IF etDiag <> GD.ET_Diag.Ok AND NOT xUpdateStructsException THEN
	xUpdateStructsException := TRUE;
	
	stUpdateStructsException.sMsg := PDL.FC_MultiConcat(i_sString1 := 'Update AddInterface: Nocke1 - ', 
														i_sString2 := GD.FC_EtDiagToString(i_etDiag := etDiag), 
														i_sString3 := ' - ', 
														i_sString4 := FC_EtDiagExtExampleLeafModuleToString(i_etDiagExt := etDiagExtExampleLeaf));
END_IF	

(*****************************************************************************************************************************************************)
(* Update ILS Data *)

// stSlave3Interface.stEndless.pstIlsData	:= ADR(G_stIlsData);
// stSlave3Interface.stMultiCam.pstIlsData	:= ADR(G_stIlsData);

// stSlave4Interface.stEndless.pstIlsData	:= ADR(G_stIlsData);
// stSlave4Interface.stMultiCam.pstIlsData	:= ADR(G_stIlsData);

(*****************************************************************************************************************************************************)
(* Set exception if any exception occurred *)

fbExceptionHandler.SetException(i_xExceptionActive	:= xUpdateStructsException, 
								iq_stException		:= stUpdateStructsException, 
								iq_stExceptionList	:= iq_stExceptionList);
					
xInitSuccessful := xInitSuccessful AND NOT xUpdateStructsException;

etDiag := GD.ET_Diag.Ok;	
(* End of system generated code, could be modified for your application *)
END_ACTION

END_PROGRAM

// LMC_PacDrive/Application/FB_ExampleLeafModule
FUNCTION_BLOCK FB_ExampleLeafModule

VAR_IN_OUT
(* TPL.ST_StandardModuleInterface *)	
	iq_stStandardModuleItf			: TPL.ST_StandardModuleInterface;
	
(* ExceptionHandling and Logging *)	
	iq_stExceptionList				: TPL.ST_ExceptionList;
	iq_stLogDataList				: TPL.ST_LogDataList;
	
(* ST_ExampleLeafModuleInterface *)
	iq_stExampleLeafModuleItf		: ST_ExampleLeafModuleInterface;
END_VAR

VAR
	xEnableFlag : BOOL;
	
	udii : UDINT;
	
	xInitHomingDone : BOOL;
	xNotAbleToSetException : BOOL;

	etDiagBuffer		: GD.ET_Diag;
	etDiagExtBufferTPL	: TPL.ET_DiagExt;
	sDiagMsgBuffer		: STRING[80];
	
	xDiagQuitFlag : BOOL;
	
	
	xExceptionReactionOutsideRange		: BOOL;
	
	stExceptionInit						: TPL.ST_Exception;
	stExceptionCmdImpossibleState		: TPL.ST_Exception;
	stExceptionCmdUnknown				: TPL.ST_Exception;
	stExceptionCmdImpossibleOverwrite	: TPL.ST_Exception;
	stWarningCmdImpossibleReaction		: TPL.ST_Exception;
	stExceptionHoming					: TPL.ST_Exception;
	stExceptionModuleReaction1			: TPL.ST_Exception;
	stExceptionModuleReaction2			: TPL.ST_Exception;
	stExceptionModuleReaction3			: TPL.ST_Exception;
	stExceptionModuleReaction4			: TPL.ST_Exception;
	stExceptionDriveFatal				: TPL.ST_Exception;
	stExcepitonDrive					: TPL.ST_Exception;
	stWarningDrive						: TPL.ST_Exception;

	stModuleReaction			: TPL.ST_Reaction;
	stLocalReaction				: TPL.ST_Reaction;
	stEmptyReaction				: TPL.ST_Reaction;
	stReaction1					: TPL.ST_Reaction;
	stReaction2					: TPL.ST_Reaction;
	stReaction3					: TPL.ST_Reaction;
	stReaction4					: TPL.ST_Reaction;

	udiDoSomethingCounter	: UDINT := 0;

	xCheckCmdException	: BOOL;
	xOpModeCmd			: BOOL;
	xCommandRefused		: BOOL;

	(* OpMode enable and active flags *)
	xHomingEnable : BOOL;
	xHomingActive : BOOL;
	xAutoEnable : BOOL;
	xAutoActive : BOOL;

	xCommandAcceptedInThisCycle : BOOL;

	xHomingException : BOOL;

	xRandomExceptionTrigger: BOOL;

	xStartFlag : BOOL;

	fbLogger : TPL.FB_Logger;
	fbLoggerPoint	: APL.FB_LoggerPoint;
	
	etStateOld : ET_ExampleLeafModuleState;
	udiMyResultSource : UDINT;
	
	ifRefActualValuesPosition : SystemConfigurationItf.IF_RefActualValuesPosition; 
	xSuccess : BOOL;
END_VAR

VAR CONSTANT
	c_udiDoSomeThingLevel : UDINT := 500;
END_VAR

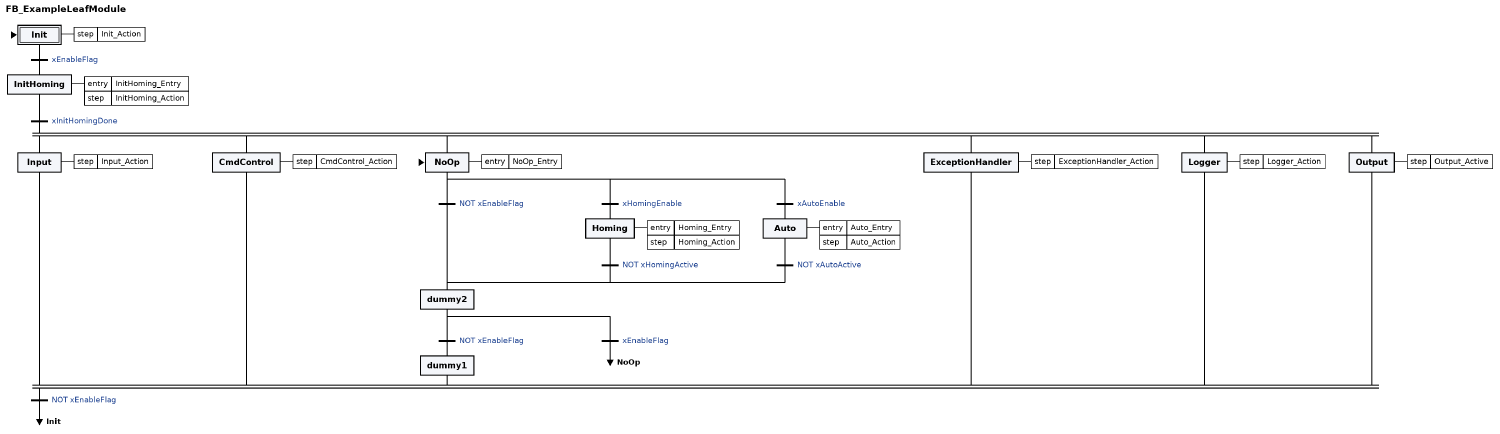
INITIAL_STEP Init:
    Init_Action(N);  // step action
END_STEP
TRANSITION FROM Init TO InitHoming
    := xEnableFlag;
END_TRANSITION
STEP InitHoming:
    InitHoming_Entry(P1);  // entry action
    InitHoming_Action(N);  // step action
END_STEP
TRANSITION FROM InitHoming TO (Input, CmdControl, NoOp, ExceptionHandler, Logger, Output)
    := xInitHomingDone;
END_TRANSITION
STEP Input:
    Input_Action(N);  // step action
END_STEP
STEP CmdControl:
    CmdControl_Action(N);  // step action
END_STEP
STEP NoOp:
    NoOp_Entry(P1);  // entry action
END_STEP
TRANSITION FROM NoOp TO dummy2
    := NOT xEnableFlag;
END_TRANSITION
TRANSITION FROM NoOp TO Homing
    := xHomingEnable;
END_TRANSITION
STEP Homing:
    Homing_Entry(P1);  // entry action
    Homing_Action(N);  // step action
END_STEP
TRANSITION FROM Homing TO dummy2
    := NOT xHomingActive;
END_TRANSITION
TRANSITION FROM NoOp TO Auto
    := xAutoEnable;
END_TRANSITION
STEP Auto:
    Auto_Entry(P1);  // entry action
    Auto_Action(N);  // step action
END_STEP
TRANSITION FROM Auto TO dummy2
    := NOT xAutoActive;
END_TRANSITION
STEP dummy2:
END_STEP
TRANSITION FROM dummy2 TO dummy1
    := NOT xEnableFlag;
END_TRANSITION
TRANSITION FROM dummy2 TO NoOp
    := xEnableFlag;
END_TRANSITION
STEP dummy1:
END_STEP
STEP ExceptionHandler:
    ExceptionHandler_Action(N);  // step action
END_STEP
STEP Logger:
    Logger_Action(N);  // step action
END_STEP
STEP Output:
    Output_Active(N);  // step action
END_STEP
TRANSITION FROM (Input, CmdControl, dummy1, ExceptionHandler, Logger, Output) TO Init
    := NOT xEnableFlag;
END_TRANSITION

ACTION Auto_Action:
(* Start application code *)
IF(iq_stExampleLeafModuleItf.q_etState = ET_ExampleLeafModuleState.AutoWaitForStart) THEN
	IF(xAutoEnable) THEN
		IF(xStartFlag) THEN
			iq_stExampleLeafModuleItf.q_etState := ET_ExampleLeafModuleState.AutoRunning;
		END_IF
	ELSE
		xAutoActive := FALSE;
	END_IF
END_IF

IF(NOT xStartFlag AND iq_stExampleLeafModuleItf.q_etState = ET_ExampleLeafModuleState.AutoRunning) THEN
	iq_stExampleLeafModuleItf.q_etState := ET_ExampleLeafModuleState.AutoWaitForStart;
END_IF

IF(iq_stExampleLeafModuleItf.q_etState = ET_ExampleLeafModuleState.AutoRunning) THEN
	IF(xAutoEnable) THEN
		iq_stExampleLeafModuleItf.q_xValue := ifRefActualValuesPosition.RefPosition >= iq_stExampleLeafModuleItf.i_lrPosMin AND 
													ifRefActualValuesPosition.RefPosition <= iq_stExampleLeafModuleItf.i_lrPosMax;
	ELSE
		iq_stExampleLeafModuleItf.q_etState := ET_ExampleLeafModuleState.AutoWaitForStart;
	END_IF
END_IF
(* End application code *)
END_ACTION

ACTION Auto_Entry:
iq_stExampleLeafModuleItf.q_etState := ET_ExampleLeafModuleState.AutoWaitForStart;
xAutoActive := TRUE;
END_ACTION

METHOD CancelException
VAR_IN_OUT
	iq_stException	: TPL.ST_Exception;
END_VAR
TPL.FC_SetException(	i_xExceptionActive	:= FALSE,
						iq_stException		:= iq_stException,
						iq_stExceptionList	:= iq_stExceptionList,
						iq_stLogDataList	:= iq_stLogDataList,
						q_etDiag 			=> etDiagBuffer,
						q_etDiagExt 		=> etDiagExtBufferTPL,
						q_sMsg 				=> sDiagMsgBuffer);
END_METHOD

ACTION CheckCmd:
(*--------------------------------------------------------------------------------------------------*)
(* CheckCMD is checking if CMD is supported by this module *)
(*--------------------------------------------------------------------------------------------------*)
xOpModeCMD			:= FALSE;
xCheckCmdException	:= FALSE;

IF 	iq_stStandardModuleItf.iq_diCMD = ET_ExampleLeafModuleCmd.Homing OR
	iq_stStandardModuleItf.iq_diCMD = ET_ExampleLeafModuleCmd.Auto OR
	iq_stStandardModuleItf.iq_diCMD = ET_ExampleLeafModuleCmd.Stop THEN

	xOpModeCMD := TRUE;
ELSIF iq_stStandardModuleItf.iq_diCMD = ET_ExampleLeafModuleCmd.Start OR
	  iq_stStandardModuleItf.iq_diCMD = ET_ExampleLeafModuleCmd.Hold THEN
	;
ELSE
	xCheckCmdException := TRUE;
END_IF
END_ACTION

ACTION CmdControl_Action:
(* CMD execution

	algorithm:
	----------

	detect new command?
		check command?
			execute command;
		end
	end

	is command running (at least one cycle)?	
		is command finished?
			signal success/unsuccessful
		end
	end
*)

xCommandAcceptedInThisCycle := FALSE;

(* Detect new command *)
IF(iq_stStandardModuleItf.i_xEnable) THEN
	IF (iq_stStandardModuleItf.iq_diCMD > 0 AND (NOT iq_stStandardModuleItf.q_xCMDActive (* In case no command is active *)
			OR iq_stStandardModuleItf.iq_diCMD <> iq_stStandardModuleItf.q_diCMDActive) (* In case a command is active *)) THEN
	
		xCommandRefused := FALSE; (* Flag is set by RefuseCommand() action *)
	
		(* Check command *)
		CheckCmd();
		IF(xCheckCmdException) THEN
			(*** Check for unknown command ***)
			stExceptionCmdUnknown.sMsg := Standard.CONCAT('Cmd unknown: ',DINT_TO_STRING(iq_stStandardModuleItf.iq_diCmd));
			ReportException(iq_stException := stExceptionCmdUnknown); 
			RefuseCommand();
		ELSE
			(*** Check for impossible overwrite ***)
			IF(iq_stStandardModuleItf.q_xCMDActive AND iq_stStandardModuleItf.iq_diCMD <> ET_ExampleLeafModuleCmd.Stop) THEN (* In this module only the ET_ExampleLeafModuleCmd.Stop command can overwrite other commands *)
				stExceptionCmdImpossibleOverwrite.sMsg := PDL.FC_MultiConcat(	i_sString1 := 'Cmd impossible: ',
																				i_sString2 := FC_EtExampleLeafModuleCmdToString(i_diCmd := iq_stStandardModuleItf.iq_diCmd),
																				i_sString3 := '; Cmd active: ',
																				i_sString4 := FC_EtExampleLeafModuleCmdToString(i_diCmd := iq_stStandardModuleItf.q_diCmdActive) );
				ReportException(iq_stException := stExceptionCmdImpossibleOverwrite);	
				RefuseCommand();
			ELSE
				(*** Check for impossible state ***)
				IF(NOT xOpModeCmd AND (* In this module, all OpMode commands are always possible independent of the state *)
					(iq_stExampleLeafModuleItf.q_etState = ET_ExampleLeafModuleState.NoOp (* Start and Hold are not possible in NoOp *)
					OR (iq_stExampleLeafModuleItf.q_etState = ET_ExampleLeafModuleState.HomingWaitForStart OR iq_stExampleLeafModuleItf.q_etState = ET_ExampleLeafModuleState.HomingDone) AND iq_stStandardModuleItf.iq_diCMD = ET_ExampleLeafModuleCmd.Hold) (* Hold is not supported in homing *)
					) THEN
					stExceptionCmdImpossibleState.sMsg := PDL.FC_MultiConcat(	i_sString1 := 'Cmd impossible: ',
																				i_sString2 := FC_EtExampleLeafModuleCmdToString(i_diCmd := iq_stStandardModuleItf.iq_diCmd),
																				i_sString3 := '; State: ',
																				i_sString4 := FC_EtExampleLeafModuleStateToString(i_etState := iq_stExampleLeafModuleItf.q_etState) );
					ReportException(iq_stException := stExceptionCmdImpossibleState);
					RefuseCommand();
				ELSE
					(* Check for impossible commands due to active error reactions *)
					IF	iq_stStandardModuleItf.iq_diCMD = ET_ExampleLeafModuleCmd.Start 
							AND (stModuleReaction.axReaction[TPL.ET_Reaction.AsyncStop] OR 
								 stModuleReaction.axReaction[TPL.ET_Reaction.SyncStopEH] OR 
								 stModuleReaction.axReaction[TPL.ET_Reaction.SyncStopEL] OR 
								 stModuleReaction.axReaction[TPL.ET_Reaction.StopEndOfCycle]) (* Start impossible if error reaction 4 or higher *)
						OR 
						
						iq_stStandardModuleItf.iq_diCMD <> ET_ExampleLeafModuleCmd.Stop 
							AND (stModuleReaction.axReaction[TPL.ET_Reaction.AsyncStop] OR 
								 stModuleReaction.axReaction[TPL.ET_Reaction.SyncStopEH] OR 
								 stModuleReaction.axReaction[TPL.ET_Reaction.SyncStopEL]) THEN (* Everything else, with exception of Stop, impossible if error reaction 3 or higher *)

						stWarningCmdImpossibleReaction.sMsg := PDL.FC_MultiConcat(	i_sString1 := 'Cmd impossible: ',
																					i_sString2 := FC_EtExampleLeafModuleCmdToString(i_diCmd := iq_stStandardModuleItf.iq_diCmd),
																					i_sString3 := '; Reaction: ',
																					i_sString4 := TPL.FC_GetStandardReactionName(iq_stReaction := stModuleReaction));
						ReportException(iq_stException := stWarningCmdImpossibleReaction);
						RefuseCommand();
					END_IF
				END_IF
			END_IF
		END_IF
	
		IF(NOT xCommandRefused) THEN (* Command has passed all checks, execute command *)
			IF fbLoggerPoint.etLogLevel >= APL.ET_LogLevel.UserAction THEN
				fbLoggerPoint.AddLogEntry(	i_etLogLevel	:= APL.ET_LogLevel.UserAction,
											i_etDiag		:= GD.ET_Diag.Ok,
											i_udiDiagExt	:= ET_DiagExtExampleLeafModule.Ok,
											i_sMessage		:= Standard.CONCAT(Standard.CONCAT(Standard.CONCAT('Command executing: ', FC_etExampleLeafModuleCmdToString(i_diCmd := iq_stStandardModuleItf.iq_diCmd)),' number: '),DINT_TO_STRING(iq_stStandardModuleItf.iq_diCmd)),
											q_etDiag		:= ,
											q_etDiagExt		:= );
			END_IF
			(* Accept command *)
			iq_stStandardModuleItf.q_xCMDActive := TRUE;
			iq_stStandardModuleItf.q_xCMDDone := FALSE;
			iq_stStandardModuleItf.q_diCMDActive := iq_stStandardModuleItf.iq_diCMD;
	
			xCommandAcceptedInThisCycle := TRUE; (* Signal for command done checks *)
	
			IF(xOpModeCMD) THEN
				DisableAllJobs();
				
				CASE iq_stStandardModuleItf.iq_diCMD OF
					ET_ExampleLeafModuleCmd.Stop:
						;	(* Do nothing, disabled OpMode flags automatically lead to NoOp *)
						
					ET_ExampleLeafModuleCmd.Homing:
						xHomingEnable := TRUE;
					
					ET_ExampleLeafModuleCmd.Auto:
						xAutoEnable := TRUE;
				END_CASE
			ELSE
				(* Action commands *)
				CASE iq_stStandardModuleItf.iq_diCMD OF
					ET_ExampleLeafModuleCmd.Start:
						xStartFlag := TRUE;
					
					ET_ExampleLeafModuleCmd.Hold:
						xStartFlag := FALSE;
				END_CASE
			END_IF
		END_IF (* New command? *)
	END_IF

(********************************************* Check successful and unsucessful of given commands ****************************************)

	(* Check if active command is done or is stopped by an error *)
	IF(NOT xCommandAcceptedInThisCycle) THEN (* Don't execute these checks if we accepted a new command in this cycle
		to ensure that execution of every command requires a minimum of 2 cycles *)

		IF(iq_stStandardModuleItf.q_xCMDActive) THEN
			CASE iq_stStandardModuleItf.iq_diCmd OF
				ET_ExampleLeafModuleCmd.Homing:
					(* Successful *)
					IF(xHomingActive) THEN
						SignalSuccessfulExecution();
					END_IF
					(* Unsucessful *)
					IF (stModuleReaction.axReaction[TPL.ET_Reaction.AsyncStop] OR 
						stModuleReaction.axReaction[TPL.ET_Reaction.SyncStopEL] OR 
						stModuleReaction.axReaction[TPL.ET_Reaction.SyncStopEH]) THEN
						
						SignalUnsuccessfulExecution();
					END_IF
					
				ET_ExampleLeafModuleCmd.Auto:
					(* Successful *)
					IF(xAutoActive) THEN
						SignalSuccessfulExecution();
					END_IF
					(* Unsucessful *)
					IF (stModuleReaction.axReaction[TPL.ET_Reaction.AsyncStop] OR 
						stModuleReaction.axReaction[TPL.ET_Reaction.SyncStopEL] OR 
						stModuleReaction.axReaction[TPL.ET_Reaction.SyncStopEH]) THEN

						SignalUnsuccessfulExecution();
					END_IF
	
				ET_ExampleLeafModuleCmd.Stop:
					(* Successful *)
					IF(iq_stExampleLeafModuleItf.q_etState = ET_ExampleLeafModuleState.NoOp) THEN
						SignalSuccessfulExecution();
					END_IF
					
				ET_ExampleLeafModuleCmd.Start:
					IF(iq_stExampleLeafModuleItf.q_etState = ET_ExampleLeafModuleState.HomingDone) THEN
						xStartFlag := FALSE;
					END_IF
					(* Successful *)
					IF(iq_stExampleLeafModuleItf.q_etState = ET_ExampleLeafModuleState.HomingDone AND NOT xHomingException
						OR iq_stExampleLeafModuleItf.q_etState = ET_ExampleLeafModuleState.AutoRunning) THEN
						SignalSuccessfulExecution();
					END_IF
					(* Unsucessful *)
					IF (stModuleReaction.axReaction[TPL.ET_Reaction.AsyncStop] OR 
						stModuleReaction.axReaction[TPL.ET_Reaction.SyncStopEL] OR 
						stModuleReaction.axReaction[TPL.ET_Reaction.SyncStopEH] OR 
						stModuleReaction.axReaction[TPL.ET_Reaction.StopEndOfCycle]  OR
						iq_stExampleLeafModuleItf.q_etState = ET_ExampleLeafModuleState.HomingDone AND xHomingException) THEN
						
						SignalUnsuccessfulExecution();
					END_IF
					
				ET_ExampleLeafModuleCmd.Hold:
					(* Successful *)
					IF(iq_stExampleLeafModuleItf.q_etState = ET_ExampleLeafModuleState.AutoWaitForStart) THEN
						SignalSuccessfulExecution();
					END_IF
					(* Unsucessful *)
					IF (stModuleReaction.axReaction[TPL.ET_Reaction.AsyncStop] OR 
						stModuleReaction.axReaction[TPL.ET_Reaction.SyncStopEL] OR 
						stModuleReaction.axReaction[TPL.ET_Reaction.SyncStopEH]) THEN

						SignalUnsuccessfulExecution();
					END_IF
			END_CASE
		END_IF
	END_IF
ELSE
	(* Module is going to be disabled *)
	iq_stStandardModuleItf.q_xReady := FALSE;
	xEnableFlag := FALSE;
	
	DisableAllJobs();
	
	xStartFlag := FALSE;

	IF(iq_stStandardModuleItf.q_xCmdActive) THEN (* If a command is currently active, cancel its execution *)
		SignalUnsuccessfulExecution();
	ELSE
		InactiveCmdExecution(); (* Command processing as if we were disabled *)
	END_IF
END_IF
END_ACTION

ACTION DiagQuit:
IF(iq_stStandardModuleItf.i_xDiagQuit AND NOT xDiagQuitFlag) THEN
	(* Rising edge of error quit *)
	xDiagQuitFlag := TRUE;
	xNotAbleToSetException := FALSE;

	FOR udii := 1 TO TPL.ET_Reaction.MainsContactorOff DO
		stLocalReaction.axReaction[udii] := FALSE;
	END_FOR

	iq_stStandardModuleItf.q_etDiag := GD.ET_Diag.Ok;

	IF(iq_stStandardModuleItf.iq_diCMD < 0) THEN
		iq_stStandardModuleItf.iq_diCMD := 0;
	END_IF
	IF fbLoggerPoint.etLogLevel >= APL.ET_LogLevel.UserAction THEN
		fbLoggerPoint.AddLogEntry(	i_etLogLevel	:= APL.ET_LogLevel.UserAction,
									i_etDiag		:= GD.ET_Diag.Ok,
									i_udiDiagExt	:= ET_DiagExtExampleLeafModule.Ok,
									i_sMessage		:= 'Diag Quit',
									q_etDiag		:= ,
									q_etDiagExt		:= );
	END_IF
ELSIF(NOT iq_stStandardModuleItf.i_xDiagQuit AND xDiagQuitFlag) THEN
	xDiagQuitFlag := FALSE;
END_IF
END_ACTION

ACTION DisableAllJobs:
(* Disable current OpMode and enable next one *)
xHomingEnable := FALSE;
xAutoEnable := FALSE;

xStartFlag := FALSE; (* On OpMode change, always reset the start flag *)
END_ACTION

ACTION Homing_Entry:
iq_stExampleLeafModuleItf.q_etState := ET_ExampleLeafModuleState.HomingWaitForStart;
xHomingActive := TRUE;


(* Start application code *)
udiDoSomethingCounter := 0;
(* End application code *)
END_ACTION

ACTION InactiveCmdExecution:
(* Command execution if module is not active (q_xActive = FALSE) or currently deactivating (i_xEnable = FALSE, q_xActive is still TRUE) *)
IF iq_stStandardModuleItf.iq_diCmd <> 0 THEN
	IF(NOT iq_stStandardModuleItf.i_xEnable) THEN
		iq_stStandardModuleItf.iq_diCmd := 0; (* All commands are signaled executed if module is disabled *)
(*ELSE*)
	ELSIF(iq_stStandardModuleItf.iq_diCmd > 0) THEN (* New command *)
		(* Command execution during enable but module is not ready for commands yet ==> error *)
		//xExceptionCmdImpossibleState := TRUE;

		stExceptionCmdImpossibleState.sMsg := PDL.FC_MultiConcat(	i_sString1 := 'Cmd impossible: ',
																	i_sString2 := FC_EtExampleLeafModuleCmdToString(i_diCmd := ABS(iq_stStandardModuleItf.iq_diCmd)),
																	i_sString3 := '; State: ',
																	i_sString4 := FC_EtExampleLeafModuleStateToString(i_etState := iq_stExampleLeafModuleItf.q_etState));
		ReportException(iq_stException := stExceptionCmdImpossibleState);
		iq_stStandardModuleItf.iq_diCmd:= - ABS(iq_stStandardModuleItf.iq_diCmd);
	END_IF
END_IF
iq_stStandardModuleItf.q_xCmdActive := FALSE;
iq_stStandardModuleItf.q_xCmdDone := FALSE;
iq_stStandardModuleItf.q_diCmdActive := 0;
END_ACTION

ACTION Init_Action:
iq_stStandardModuleItf.q_xActive			:= FALSE;
iq_stStandardModuleItf.q_xReady				:= FALSE;

iq_stStandardModuleItf.q_etDiag				:= GD.ET_Diag.Ok;
iq_stStandardModuleItf.q_udiDiagExt			:= ET_DiagExtExampleLeafModule.Disabled;
iq_stStandardModuleItf.q_sDiagExt			:= FC_EtDiagExtExampleLeafModuleToString(i_etDiagExt := iq_stStandardModuleItf.q_udiDiagExt);
iq_stStandardModuleItf.q_sMsg				:= '';

iq_stStandardModuleItf.q_dwModuleType		:= ET_ModuleType.ExampleLeafModule;
iq_stStandardModuleItf.q_sModuleTypeName	:= 'ExampleLeafModule';
iq_stStandardModuleItf.q_udiModuleVersion	:= 1;

iq_stExampleLeafModuleItf.q_etState	:= ET_ExampleLeafModuleState.Disabled;

THIS^.DiagQuit();
THIS^.InactiveCmdExecution();

udiMyResultSource := ET_ExceptionSource.ExampleLeafModule; (* Has to be coded this way to get around compiler restrictions*)

(* detect invalid configurations and avoid array index out of range error *)
IF(iq_stStandardModuleItf.iq_stExt.udiReactionOffset + TPL. ET_Reaction.MainsContactorOff > TPL.Gc_udiMaxNumberOfReactions) OR xExceptionReactionOutsideRange THEN (* module uses error reactions 1 to 5 *)
	xExceptionReactionOutsideRange := TRUE; (* create unquittable error *)
	
	(* create exception *)
	stExceptionInit.etDiag					:= GD.ET_Diag.InputParameterInvalid;
	stExceptionInit.udiDiagExt				:= ET_DiagExtExampleLeafModule.ReactionOffsetRange;
	stExceptionInit.sMsg					:= Standard.CONCAT('Value: ', UDINT_TO_STRING(iq_stStandardModuleItf.iq_stExt.udiReactionOffset));
	stExceptionInit.udiModuleId				:= iq_stStandardModuleItf.i_udiModuleId;
	stExceptionInit.sModuleName				:= iq_stStandardModuleItf.i_sModuleName;
	stExceptionInit.etSource				:= udiMyResultSource;
	stExceptionInit.timDelayTime			:= T#0MS;
	stExceptionInit.wHmiAttributes			:= 0;
	stExceptionInit.xAutoQuit				:= FALSE;
	stExceptionInit.stReaction.axReaction[TPL.ET_Reaction.AsyncStop]	:= TRUE; (* without offset on purpose *)
	
	iq_stStandardModuleItf.iq_stExt.udiReactionOffset := 0;
	
	ReportException(iq_stException := stExceptionInit);
ELSIF (iq_stStandardModuleItf.i_xEnable) THEN
	stReaction1 := stEmptyReaction;
	stReaction1.axReaction[iq_stStandardModuleItf.iq_stExt.udiReactionOffset + TPL.ET_Reaction.AsyncStop] := TRUE;
	stReaction2 := stEmptyReaction;
	stReaction2.axReaction[iq_stStandardModuleItf.iq_stExt.udiReactionOffset + TPL.ET_Reaction.SyncStopEL] := TRUE;
	stReaction3 := stEmptyReaction;
	stReaction3.axReaction[iq_stStandardModuleItf.iq_stExt.udiReactionOffset + TPL.ET_Reaction.SyncStopEH] := TRUE;
	stReaction4 := stEmptyReaction;
	stReaction4.axReaction[iq_stStandardModuleItf.iq_stExt.udiReactionOffset + TPL.ET_Reaction.StopEndOfCycle] := TRUE;
	
	(* Initialization of exception structures *)
	stExceptionCmdUnknown.etDiag						:= GD.ET_Diag.ExecutionAborted;
	stExceptionCmdUnknown.udiDiagExt					:= ET_DiagExtExampleLeafModule.CmdUnknown;
	stExceptionCmdUnknown.sMsg							:= 'Command unknown'; (* Replaced on usage *)
	stExceptionCmdUnknown.udiModuleId					:= iq_stStandardModuleItf.i_udiModuleId;
	stExceptionCmdUnknown.sModuleName					:= iq_stStandardModuleItf.i_sModuleName;
	stExceptionCmdUnknown.etSource						:= udiMyResultSource;
	stExceptionCmdUnknown.timDelayTime					:= T#0MS;
	stExceptionCmdUnknown.wHmiAttributes				:= 0;
	stExceptionCmdUnknown.xAutoQuit						:= FALSE;
	stExceptionCmdUnknown.stReaction					:= stReaction1;

	stExceptionCmdImpossibleOverwrite.etDiag			:= GD.ET_Diag.ExecutionAborted;
	stExceptionCmdImpossibleOverwrite.udiDiagExt		:= ET_DiagExtExampleLeafModule.CmdImpossibleOverwrite;
	stExceptionCmdImpossibleOverwrite.sMsg				:= 'Impossible command overwrite'; (* Replaced on usage *)
	stExceptionCmdImpossibleOverwrite.udiModuleId		:= iq_stStandardModuleItf.i_udiModuleId;
	stExceptionCmdImpossibleOverwrite.sModuleName		:= iq_stStandardModuleItf.i_sModuleName;
	stExceptionCmdImpossibleOverwrite.etSource			:= udiMyResultSource;
	stExceptionCmdImpossibleOverwrite.timDelayTime		:= T#0MS;
	stExceptionCmdImpossibleOverwrite.wHmiAttributes	:= 0;
	stExceptionCmdImpossibleOverwrite.xAutoQuit			:= FALSE;
	stExceptionCmdImpossibleOverwrite.stReaction		:= stReaction1;
	
	stExceptionCmdImpossibleState.etDiag				:= GD.ET_Diag.ExecutionAborted;
	stExceptionCmdImpossibleState.udiDiagExt			:= ET_DiagExtExampleLeafModule.CmdImpossibleState;
	stExceptionCmdImpossibleState.sMsg					:= 'Impossible command for state'; (* Replaced on usage *)
	stExceptionCmdImpossibleState.udiModuleId			:= iq_stStandardModuleItf.i_udiModuleId;
	stExceptionCmdImpossibleState.sModuleName			:= iq_stStandardModuleItf.i_sModuleName;
	stExceptionCmdImpossibleState.etSource				:= udiMyResultSource;
	stExceptionCmdImpossibleState.timDelayTime			:= T#0MS;
	stExceptionCmdImpossibleState.wHmiAttributes		:= 0;
	stExceptionCmdImpossibleState.xAutoQuit				:= FALSE;
	stExceptionCmdImpossibleState.stReaction			:= stReaction1;

	stWarningCmdImpossibleReaction.etDiag				:= GD.ET_Diag.ExecutionAborted;
	stWarningCmdImpossibleReaction.udiDiagExt			:= ET_DiagExtExampleLeafModule.CmdImpossibleReaction;
	stWarningCmdImpossibleReaction.sMsg					:= 'Impossible command on reaction'; (* Replaced on usage *)
	stWarningCmdImpossibleReaction.udiModuleId			:= iq_stStandardModuleItf.i_udiModuleId;
	stWarningCmdImpossibleReaction.sModuleName			:= iq_stStandardModuleItf.i_sModuleName;
	stWarningCmdImpossibleReaction.etSource				:= udiMyResultSource;
	stWarningCmdImpossibleReaction.timDelayTime			:= T#0MS;
	stWarningCmdImpossibleReaction.wHmiAttributes		:= 0;
	stWarningCmdImpossibleReaction.xAutoQuit			:= FALSE;
	
	stExceptionModuleReaction1.etDiag					:= GD.ET_Diag.InputParameterInvalid;(* Replaced on usage *)
	stExceptionModuleReaction1.udiDiagExt				:= ET_DiagExtExampleLeafModule.Ok;(* Replaced on usage *)
	stExceptionModuleReaction1.sMsg						:= '';(* Replaced on usage *)
	stExceptionModuleReaction1.udiModuleId				:= iq_stStandardModuleItf.i_udiModuleId;
	stExceptionModuleReaction1.sModuleName				:= iq_stStandardModuleItf.i_sModuleName;
	stExceptionModuleReaction1.etSource					:= udiMyResultSource;
	stExceptionModuleReaction1.timDelayTime				:= T#0MS;
	stExceptionModuleReaction1.wHmiAttributes			:= 0;
	stExceptionModuleReaction1.xAutoQuit				:= FALSE;
	stExceptionModuleReaction1.stReaction				:= stReaction1;

	stExceptionModuleReaction2.etDiag					:= GD.ET_Diag.InputParameterInvalid;(* Replaced on usage *)
	stExceptionModuleReaction2.udiDiagExt				:= ET_DiagExtExampleLeafModule.Ok;(* Replaced on usage *)
	stExceptionModuleReaction2.sMsg						:= '';(* Replaced on usage *)
	stExceptionModuleReaction2.udiModuleId				:= iq_stStandardModuleItf.i_udiModuleId;
	stExceptionModuleReaction2.sModuleName				:= iq_stStandardModuleItf.i_sModuleName;
	stExceptionModuleReaction2.etSource					:= udiMyResultSource;
	stExceptionModuleReaction2.timDelayTime				:= T#0MS;
	stExceptionModuleReaction2.wHmiAttributes			:= 0;
	stExceptionModuleReaction2.xAutoQuit				:= FALSE;
	stExceptionModuleReaction2.stReaction				:= stReaction2;

	stExceptionModuleReaction3.etDiag					:= GD.ET_Diag.InputParameterInvalid;(* Replaced on usage *)
	stExceptionModuleReaction3.udiDiagExt				:= ET_DiagExtExampleLeafModule.Ok;(* Replaced on usage *)
	stExceptionModuleReaction3.sMsg						:= '';(* Replaced on usage *)
	stExceptionModuleReaction3.udiModuleId				:= iq_stStandardModuleItf.i_udiModuleId;
	stExceptionModuleReaction3.sModuleName				:= iq_stStandardModuleItf.i_sModuleName;
	stExceptionModuleReaction3.etSource					:= udiMyResultSource;
	stExceptionModuleReaction3.timDelayTime				:= T#0MS;
	stExceptionModuleReaction3.wHmiAttributes			:= 0;
	stExceptionModuleReaction3.xAutoQuit				:= FALSE;
	stExceptionModuleReaction3.stReaction				:= stReaction3;

	stExceptionModuleReaction4.etDiag					:= GD.ET_Diag.InputParameterInvalid;(* Replaced on usage *)
	stExceptionModuleReaction4.udiDiagExt				:= ET_DiagExtExampleLeafModule.Ok;(* Replaced on usage *)
	stExceptionModuleReaction4.sMsg						:= '';(* Replaced on usage *)
	stExceptionModuleReaction4.udiModuleId				:= iq_stStandardModuleItf.i_udiModuleId;
	stExceptionModuleReaction4.sModuleName				:= iq_stStandardModuleItf.i_sModuleName;
	stExceptionModuleReaction4.etSource					:= udiMyResultSource;
	stExceptionModuleReaction4.timDelayTime				:= T#0MS;
	stExceptionModuleReaction4.wHmiAttributes			:= 0;
	stExceptionModuleReaction4.xAutoQuit				:= FALSE;
	stExceptionModuleReaction4.stReaction				:= stReaction4;
	
	stExceptionDriveFatal.etDiag						:= GD.ET_Diag.DriveConditionInvalid;
	stExceptionDriveFatal.udiDiagExt					:= ET_DiagExtExampleLeafModule.DriveFatalException;
	stExceptionDriveFatal.sMsg							:= 'Drive diag'; (* Replaced on usage *)
	stExceptionDriveFatal.udiModuleId					:= iq_stStandardModuleItf.i_udiModuleId;
	stExceptionDriveFatal.sModuleName					:= iq_stStandardModuleItf.i_sModuleName;
	stExceptionDriveFatal.etSource						:= udiMyResultSource;
	stExceptionDriveFatal.timDelayTime					:= T#0MS;
	stExceptionDriveFatal.wHmiAttributes				:= 0;
	stExceptionDriveFatal.xAutoQuit						:= FALSE;
	stExceptionDriveFatal.stReaction					:= stReaction1;
	
	stExcepitonDrive.etDiag								:= GD.ET_Diag.DriveConditionInvalid;
	stExcepitonDrive.udiDiagExt							:= ET_DiagExtExampleLeafModule.DriveException;
	stExcepitonDrive.sMsg								:= 'Drive diag'; (* Replaced on usage *)
	stExcepitonDrive.udiModuleId						:= iq_stStandardModuleItf.i_udiModuleId;
	stExcepitonDrive.sModuleName						:= iq_stStandardModuleItf.i_sModuleName;
	stExcepitonDrive.etSource							:= udiMyResultSource;
	stExcepitonDrive.timDelayTime						:= T#0MS;
	stExcepitonDrive.wHmiAttributes						:= 0;
	stExcepitonDrive.xAutoQuit							:= FALSE;
	stExcepitonDrive.stReaction							:= stReaction2;

	stWarningDrive.etDiag								:= GD.ET_Diag.DriveConditionInvalid;
	stWarningDrive.udiDiagExt							:= ET_DiagExtExampleLeafModule.DriveWarning;
	stWarningDrive.sMsg									:= 'Drive warning'; (* Replaced on usage *)
	stWarningDrive.udiModuleId							:= iq_stStandardModuleItf.i_udiModuleId;
	stWarningDrive.sModuleName							:= iq_stStandardModuleItf.i_sModuleName;
	stWarningDrive.etSource								:= udiMyResultSource;
	stWarningDrive.timDelayTime							:= T#0MS;
	stWarningDrive.wHmiAttributes						:= 0;
	stWarningDrive.xAutoQuit							:= FALSE;
	stWarningDrive.stReaction							:= stReaction4;

	stExceptionInit.etDiag								:= GD.ET_Diag.InputParameterInvalid; (* Replaced on usage *)
	stExceptionInit.udiDiagExt							:= ET_DiagExtExampleLeafModule.Ok; (* Replaced on usage *)
	stExceptionInit.sMsg								:= ''; (* Replaced on usage *)
	stExceptionInit.udiModuleId							:= iq_stStandardModuleItf.i_udiModuleId;
	stExceptionInit.sModuleName							:= iq_stStandardModuleItf.i_sModuleName;
	stExceptionInit.etSource							:= udiMyResultSource;
	stExceptionInit.timDelayTime						:= T#0MS;
	stExceptionInit.wHmiAttributes						:= 0;
	stExceptionInit.xAutoQuit							:= FALSE;
	stExceptionInit.stReaction							:= stReaction1;
	
	stExceptionHoming.etDiag							:= GD.ET_Diag.HomingFailed;
	stExceptionHoming.udiDiagExt						:= ET_DiagExtExampleLeafModule.RandomException;
	stExceptionHoming.sMsg								:= '';
	stExceptionHoming.udiModuleId						:= iq_stStandardModuleItf.i_udiModuleId;
	stExceptionHoming.sModuleName						:= iq_stStandardModuleItf.i_sModuleName;
	stExceptionHoming.etSource							:= udiMyResultSource;
	stExceptionHoming.timDelayTime						:= T#0MS;
	stExceptionHoming.wHmiAttributes					:= 0;
	stExceptionHoming.xAutoQuit							:= FALSE;
	stExceptionHoming.stReaction						:= stReaction4;

	IF (iq_stExampleLeafModuleItf.i_ifDrive = 0) THEN
		stExceptionModuleReaction1.etDiag		:= GD.ET_Diag.InputParameterInvalid;
		stExceptionModuleReaction1.udiDiagExt	:= ET_DiagExtExampleLeafModule.DriveInvalid;
		stExceptionModuleReaction1.sMsg			:= 'No drive given';
		
		ReportException(iq_stException := stExceptionModuleReaction1);
	ELSE
		xEnableFlag := TRUE;
		iq_stStandardModuleItf.q_xActive := TRUE;
		
		FOR udii := 1 TO TPL.Gc_udiMaxNumberOfReactions DO
			stLocalReaction.axReaction[udii] := FALSE;
		END_FOR
		
		THIS^.SetInterfaces();
		
		xInitHomingDone := FALSE;
		
		iq_stExampleLeafModuleItf.q_etState := ET_ExampleLeafModuleState.Initializing;
		
		iq_stStandardModuleItf.q_etDiag		:= GD.ET_Diag.Ok;
		iq_stStandardModuleItf.q_udiDiagExt	:= ET_DiagExtExampleLeafModule.Initializing;
		iq_stStandardModuleItf.q_sDiagExt	:= FC_EtDiagExtExampleLeafModuleToString(ET_DiagExtExampleLeafModule.Initializing);
		iq_stStandardModuleItf.q_sMsg		:= '';
		
		IF fbLoggerPoint.etLogLevel >= APL.ET_LogLevel.UserAction THEN
			fbLoggerPoint.AddLogEntry(	i_etLogLevel	:= APL.ET_LogLevel.UserAction,
										i_etDiag		:= GD.ET_Diag.Ok,
										i_udiDiagExt	:= ET_DiagExtExampleLeafModule.Ok,
										i_sMessage		:= 'enabeling Module',
										q_etDiag		:= ,
										q_etDiagExt		:= );
		END_IF
	END_IF

END_IF

THIS^.SetOutputs();
END_ACTION

ACTION InitHoming_Action:
DiagQuit();
InactiveCmdExecution();

(* Emulating an initialization that takes some time *)
udiDoSomethingCounter := udiDoSomethingCounter + 1;
IF(iq_stExampleLeafModuleItf.i_xInitHoming) THEN
	xInitHomingDone := FALSE;
	iq_stExampleLeafModuleItf.q_xValue := TRUE;
	IF(udiDoSomethingCounter > c_udiDoSomeThingLevel) THEN
		(* Initial homing done *)
		xInitHomingDone := TRUE;
		iq_stExampleLeafModuleItf.q_xValue := TRUE;
		IF fbLoggerPoint.etLogLevel >= APL.ET_LogLevel.StatusMessage THEN
			fbLoggerPoint.AddLogEntry(	i_etLogLevel	:= APL.ET_LogLevel.StatusMessage,
										i_etDiag		:= GD.ET_Diag.Ok,
										i_udiDiagExt	:= ET_DiagExtExampleLeafModule.Ok,
										i_sMessage		:= 'InitHoming done',
										q_etDiag		:= ,
										q_etDiagExt		:= );
		END_IF
	END_IF
ELSE
	xInitHomingDone := TRUE;
END_IF

THIS^.SetOutputs();
END_ACTION

ACTION InitHoming_Entry:
udiDoSomethingCounter := 0;
END_ACTION

ACTION Input_Action:
iq_stStandardModuleItf.q_xReady := TRUE;
THIS^.DiagQuit();

(* -----------------------------------------------------------------------------------------------*)
(* Check external Reaction *)
(* -----------------------------------------------------------------------------------------------*)
stModuleReaction.axReaction[TPL.ET_Reaction.AsyncStop] := stLocalReaction.axReaction[TPL.ET_Reaction.AsyncStop] OR iq_stStandardModuleItf.i_stReaction.axReaction[TPL.ET_Reaction.AsyncStop];
stModuleReaction.axReaction[TPL.ET_Reaction.SyncStopEL] := stLocalReaction.axReaction[TPL.ET_Reaction.SyncStopEL] OR iq_stStandardModuleItf.i_stReaction.axReaction[TPL.ET_Reaction.SyncStopEL];
stModuleReaction.axReaction[TPL.ET_Reaction.SyncStopEH] := stLocalReaction.axReaction[TPL.ET_Reaction.SyncStopEH] OR iq_stStandardModuleItf.i_stReaction.axReaction[TPL.ET_Reaction.SyncStopEH];
stModuleReaction.axReaction[TPL.ET_Reaction.StopEndOfCycle] := stLocalReaction.axReaction[TPL.ET_Reaction.StopEndOfCycle] OR iq_stStandardModuleItf.i_stReaction.axReaction[TPL.ET_Reaction.StopEndOfCycle];
stModuleReaction.axReaction[TPL.ET_Reaction.MainsContactorOff] := stLocalReaction.axReaction[TPL.ET_Reaction.MainsContactorOff] OR iq_stStandardModuleItf.i_stReaction.axReaction[TPL.ET_Reaction.MainsContactorOff];
END_ACTION

ACTION NoOp_Entry:
iq_stExampleLeafModuleItf.q_etState := ET_ExampleLeafModuleState.NoOp;
END_ACTION

ACTION Output_Active:
(* System generated code, to be changed by experienced programmers *)
THIS^.SetOutputs();
(* End of system generated code, to be changed by experienced programmers *)
END_ACTION

ACTION RefuseCommand:
iq_stStandardModuleItf.q_xCMDActive := FALSE;
iq_stStandardModuleItf.q_xCMDDone := FALSE;
iq_stStandardModuleItf.iq_diCMD := - iq_stStandardModuleItf.iq_diCMD;

xCommandRefused := TRUE;
END_ACTION

METHOD PUBLIC RegisterLoggerPoint
VAR_INPUT
	i_ifParent		: APL.IF_LoggerPoint;
	i_sName			: STRING[80];
END_VAR
VAR_OUTPUT
	q_etDiag		: GD.ET_Diag := GD.ET_Diag.Ok;
	q_etDiagExt		: ET_DiagExtExampleLeafModule := ET_DiagExtExampleLeafModule.Ok;
	q_sMsg			: STRING[80] := '';
END_VAR
VAR
	etDiagBuffer		: GD.ET_Diag;
	etDiagExtBufferAPL	: APL.ET_DiagExt;
END_VAR
THIS^.fbLoggerPoint.RegisterLoggerPoint(	i_ifParent		:= i_ifParent,
											i_sName			:= i_sName,
											i_sType			:= 'FB_ExampleLeafModule',
											i_sSource		:= 'Project',
											q_etDiag		=> etDiagBuffer,
											q_etDiagExt		=> etDiagExtBufferAPL);
IF (etDiagBuffer <> GD.ET_Diag.Ok) THEN
	CASE etDiagExtBufferAPL OF
		APL.ET_DiagExt.ParentInvalid:
			q_etDiag := GD.ET_Diag.InputParameterInvalid;
			q_etDiagExt := ET_DiagExtExampleLeafModule.ParentInvalid;
			
		APL.ET_DiagExt.ParentNotRegistered:
			q_etDiag := GD.ET_Diag.InputParameterInvalid;
			q_etDiagExt := ET_DiagExtExampleLeafModule.ParentNotRegistered;
			
		APL.ET_DiagExt.MaxNumberOfLoggerPointsExeeded:
			q_etDiag := GD.ET_Diag.InputParameterInvalid;
			q_etDiagExt := ET_DiagExtExampleLeafModule.MaxNumberOfLoggerPointsExeeded;
			
	ELSE
		q_etDiag := GD.ET_Diag.UnexpectedProgramBehavior;
		q_etdiagExt := ET_DiagExtExampleLeafModule.UnexpectedDiagExt;
		q_sMsg := Standard.CONCAT('RegisterLoggerPoint: ', APL.FC_EtDiagExtToString(i_etDiagExt := etDiagExtBufferAPL));
	END_CASE
END_IF
END_METHOD

METHOD ReportException
VAR_IN_OUT
	iq_stException	: TPL.ST_Exception;
END_VAR
VAR CONSTANT
	c_diMaxReaction	: DINT := 4;
END_VAR
IF (fbLoggerPoint.etLogLevel >= APL.ET_LogLevel.CriticalException) AND (iq_stException.etDiag = GD.ET_Diag.UnexpectedProgramBehavior) THEN
	IF NOT TPL.FC_CheckExceptionIsInList( iq_stException := iq_stException, iq_stExceptionList := THIS^.iq_stExceptionList) THEN
		fbLoggerPoint.AddLogEntry(	i_etLogLevel	:= APL.ET_LogLevel.CriticalException,
									i_etDiag		:= GD.ET_Diag.Ok,
									i_udiDiagExt	:= ET_DiagExtExampleLeafModule.Ok,
									i_sMessage		:= Standard.CONCAT(Standard.CONCAT(Standard.CONCAT(Standard.CONCAT(Standard.CONCAT(Standard.CONCAT('Exception ET_Diag: ',GD.FC_EtDiagToString(i_etDiag := iq_stException.etDiag)),' ET_DiagExt: '),FC_EtDiagExtToString(i_etDiagExt := iq_stException.udiDiagExt)),' sMsg: '),iq_stException.sMsg),TPL.FC_GetStandardReactionName(iq_stReaction := iq_stException.stReaction)),
									q_etDiag		:= ,
									q_etDiagExt		:= );
	END_IF
ELSIF (fbLoggerPoint.etLogLevel >= APL.ET_LogLevel.Exception) THEN
	IF NOT TPL.FC_CheckExceptionIsInList( iq_stException := iq_stException, iq_stExceptionList := THIS^.iq_stExceptionList) THEN
		fbLoggerPoint.AddLogEntry(	i_etLogLevel	:= APL.ET_LogLevel.Exception,
									i_etDiag		:= GD.ET_Diag.Ok,
									i_udiDiagExt	:= ET_DiagExtExampleLeafModule.Ok,
									i_sMessage		:= Standard.CONCAT(Standard.CONCAT(Standard.CONCAT(Standard.CONCAT(Standard.CONCAT(Standard.CONCAT('Exception ET_Diag: ',GD.FC_EtDiagToString(i_etDiag := iq_stException.etDiag)),' ET_DiagExt: '),FC_EtDiagExtToString(i_etDiagExt := iq_stException.udiDiagExt)),' sMsg: '),iq_stException.sMsg),TPL.FC_GetStandardReactionName(iq_stReaction := iq_stException.stReaction)),
									q_etDiag		:= ,
									q_etDiagExt		:= );
	END_IF
END_IF

iq_stException.sDiagExt := FC_EtDiagExtExampleLeafModuleToString(i_etDiagExt := iq_stException.udiDiagExt);
TPL.FC_SetException(	i_xExceptionActive	:= TRUE,
						iq_stException		:= iq_stException,
						iq_stExceptionList	:= iq_stExceptionList,
						iq_stLogDataList	:= iq_stLogDataList,
						q_etDiag 			=> etDiagBuffer,
						q_etDiagExt 		=> etDiagExtBufferTPL,
						q_sMsg 				=> sDiagMsgBuffer);
						
IF (etDiagBuffer <> GD.ET_Diag.Ok) THEN
	(* if exception could not be reported, show exception on outputs *)
	xNotAbleToSetException := TRUE;
	iq_stStandardModuleItf.q_etDiag := iq_stException.etDiag;
	iq_stStandardModuleItf.q_udiDiagExt := iq_stException.udiDiagExt;
	iq_stStandardModuleItf.q_sDiagExt := iq_stException.sDiagExt;
	iq_stStandardModuleItf.q_sMsg := iq_stException.sMsg;
END_IF

stLocalReaction.axReaction[TPL.ET_Reaction.MainsContactorOff] := stLocalReaction.axReaction[TPL.ET_Reaction.MainsContactorOff] OR iq_stException.stReaction.axReaction[TPL.ET_Reaction.MainsContactorOff];
stLocalReaction.axReaction[TPL.ET_Reaction.AsyncStop] := stLocalReaction.axReaction[TPL.ET_Reaction.AsyncStop] OR iq_stException.stReaction.axReaction[TPL.ET_Reaction.AsyncStop];
stLocalReaction.axReaction[TPL.ET_Reaction.SyncStopEH] := stLocalReaction.axReaction[TPL.ET_Reaction.SyncStopEH] OR iq_stException.stReaction.axReaction[TPL.ET_Reaction.SyncStopEH];
stLocalReaction.axReaction[TPL.ET_Reaction.SyncStopEL] := stLocalReaction.axReaction[TPL.ET_Reaction.SyncStopEL] OR iq_stException.stReaction.axReaction[TPL.ET_Reaction.SyncStopEL];
(* special handling for StopEndOfCycle. Wait till reaction feedback from machine. User can transform this reaction and make own reaction.
stLocalReaction.axReaction[TPL.ET_Reaction.StopEndOfCycle] := stLocalReaction.axReaction[TPL.ET_Reaction.StopEndOfCycle] OR iq_stException.stReaction.axReaction[TPL.ET_Reaction.StopEndOfCycle];
*)

stModuleReaction.axReaction[TPL.ET_Reaction.MainsContactorOff] := stLocalReaction.axReaction[TPL.ET_Reaction.MainsContactorOff] OR stModuleReaction.axReaction[TPL.ET_Reaction.MainsContactorOff];
stModuleReaction.axReaction[TPL.ET_Reaction.AsyncStop] := stLocalReaction.axReaction[TPL.ET_Reaction.AsyncStop] OR stModuleReaction.axReaction[TPL.ET_Reaction.AsyncStop];
stModuleReaction.axReaction[TPL.ET_Reaction.SyncStopEH] := stLocalReaction.axReaction[TPL.ET_Reaction.SyncStopEH] OR stModuleReaction.axReaction[TPL.ET_Reaction.SyncStopEH];
stModuleReaction.axReaction[TPL.ET_Reaction.SyncStopEL] := stLocalReaction.axReaction[TPL.ET_Reaction.SyncStopEL] OR stModuleReaction.axReaction[TPL.ET_Reaction.SyncStopEL];
(* special handling for StopEndOfCycle. Wait till reaction feedback from machine. User can transform this reaction and make own reaction.
stModuleReaction.axReaction[TPL.ET_Reaction.StopEndOfCycle] := stLocalReaction.axReaction[TPL.ET_Reaction.StopEndOfCycle] OR stModuleReaction.axReaction[TPL.ET_Reaction.StopEndOfCycle];
*)
END_METHOD

METHOD SetOutputs
VAR_INPUT
END_VAR
IF xNotAbleToSetException THEN
	; (* Do nothing. Diag outputs show not reportable exception *)
	iq_stStandardModuleItf.q_xReady := FALSE;
ELSIF stModuleReaction.axReaction[TPL.ET_Reaction.AsyncStop] THEN
	iq_stStandardModuleItf.q_etDiag := GD.ET_Diag.ExecutionAborted;
	iq_stStandardModuleItf.q_udiDiagExt := ET_DiagExtExampleLeafModule.AsyncStop;
	iq_stStandardModuleItf.q_sDiagExt := 'AsyncStop';
	iq_stStandardModuleItf.q_sMsg := '';
	
	iq_stStandardModuleItf.q_xReady := FALSE;
ELSIF stModuleReaction.axReaction[TPL.ET_Reaction.SyncStopEL] THEN
	iq_stStandardModuleItf.q_etDiag := GD.ET_Diag.ExecutionAborted;
	iq_stStandardModuleItf.q_udiDiagExt := ET_DiagExtExampleLeafModule.SyncStopEL;
	iq_stStandardModuleItf.q_sDiagExt := 'SyncStopEL';
	iq_stStandardModuleItf.q_sMsg := '';
	
	iq_stStandardModuleItf.q_xReady := FALSE;
ELSIF stModuleReaction.axReaction[TPL.ET_Reaction.SyncStopEH] THEN
	iq_stStandardModuleItf.q_etDiag := GD.ET_Diag.ExecutionAborted;
	iq_stStandardModuleItf.q_udiDiagExt := ET_DiagExtExampleLeafModule.SyncStopEH;
	iq_stStandardModuleItf.q_sDiagExt := 'SyncStopEH';
	iq_stStandardModuleItf.q_sMsg := '';
	
	iq_stStandardModuleItf.q_xReady := FALSE;
ELSIF stModuleReaction.axReaction[TPL.ET_Reaction.StopEndOfCycle] THEN
	iq_stStandardModuleItf.q_etDiag := GD.ET_Diag.ExecutionAborted;
	iq_stStandardModuleItf.q_udiDiagExt := ET_DiagExtExampleLeafModule.StopEndOfCycle;
	iq_stStandardModuleItf.q_sDiagExt := 'StopEndOfCycle';
	iq_stStandardModuleItf.q_sMsg := '';
	
	iq_stStandardModuleItf.q_xReady := FALSE;
ELSE
	IF (iq_stExampleLeafModuleItf.q_etState <> ET_ExampleLeafModuleState.Disabled) AND
	   (iq_stExampleLeafModuleItf.q_etState <> ET_ExampleLeafModuleState.Initializing) THEN

		iq_stStandardModuleItf.q_xReady := TRUE;
	ELSE
		iq_stStandardModuleItf.q_xReady := FALSE;
	END_IF
		
	iq_stStandardModuleItf.q_etDiag := GD.ET_Diag.Ok;
	CASE iq_stExampleLeafModuleItf.q_etState OF
		ET_ExampleLeafModuleState.NoOp: 
			iq_stStandardModuleItf.q_udiDiagExt := ET_DiagExtExampleLeafModule.NoOp;
		ET_ExampleLeafModuleState.Disabled:
			iq_stStandardModuleItf.q_udiDiagExt := ET_DiagExtExampleLeafModule.Disabled;
		ET_ExampleLeafModuleState.Initializing:
			iq_stStandardModuleItf.q_udiDiagExt := ET_DiagExtExampleLeafModule.Initializing;
		ET_ExampleLeafModuleState.HomingWaitForStart:
			iq_stStandardModuleItf.q_udiDiagExt := ET_DiagExtExampleLeafModule.HomingWaitForStart;
		ET_ExampleLeafModuleState.HomingExecuting:
			iq_stStandardModuleItf.q_udiDiagExt := ET_DiagExtExampleLeafModule.HomingExecuting;
		ET_ExampleLeafModuleState.HomingDone:
			iq_stStandardModuleItf.q_udiDiagExt := ET_DiagExtExampleLeafModule.HomingDone;
		ET_ExampleLeafModuleState.AutoWaitForStart:
			iq_stStandardModuleItf.q_udiDiagExt := ET_DiagExtExampleLeafModule.AutoWaitForStart;
		ET_ExampleLeafModuleState.AutoRunning:
			iq_stStandardModuleItf.q_udiDiagExt := ET_DiagExtExampleLeafModule.AutoRunning;
	END_CASE
	iq_stStandardModuleItf.q_sDiagExt := FC_EtDiagExtExampleLeafModuleToString(i_etDiagExt := iq_stStandardModuleItf.q_udiDiagExt);
	iq_stStandardModuleItf.q_sMsg := '';
END_IF

IF fbLoggerPoint.etLogLevel >= APL.ET_LogLevel.StatusMessage THEN
	IF (iq_stExampleLeafModuleItf.q_etState <> etStateOld) THEN
		fbLoggerPoint.AddLogEntry(	i_etLogLevel	:= APL.ET_LogLevel.StatusMessage,
									i_etDiag		:= GD.ET_Diag.Ok,
									i_udiDiagExt	:= ET_DiagExtExampleLeafModule.Ok,
									i_sMessage		:= Standard.CONCAT('State changed to: ', FC_EtExampleLeafModuleStateToString(i_etState := iq_stExampleLeafModuleItf.q_etState)),
									q_etDiag		:= ,
									q_etDiagExt		:= );
	END_IF
	etStateOld := iq_stExampleLeafModuleItf.q_etState;
END_IF
END_METHOD

ACTION SignalSuccessfulExecution:
IF fbLoggerPoint.etLogLevel >= APL.ET_LogLevel.StatusMessage THEN
	fbLoggerPoint.AddLogEntry(	i_etLogLevel	:= APL.ET_LogLevel.StatusMessage,
								i_etDiag		:= GD.ET_Diag.Ok,
								i_udiDiagExt	:= ET_DiagExtExampleLeafModule.Ok,
								i_sMessage		:= Standard.CONCAT(Standard.CONCAT(Standard.CONCAT('Command done: ', FC_etExampleLeafModuleCmdToString(i_diCmd := iq_stStandardModuleItf.iq_diCmd)),' number: '),DINT_TO_STRING(iq_stStandardModuleItf.iq_diCmd)),
								q_etDiag		:= ,
								q_etDiagExt		:= );
END_IF

iq_stStandardModuleItf.q_xCMDActive := FALSE;
iq_stStandardModuleItf.q_xCMDDone := TRUE;
IF(iq_stStandardModuleItf.iq_diCMD = iq_stStandardModuleItf.q_diCMDActive) THEN
	iq_stStandardModuleItf.iq_diCMD := 0;
(* ELSE don't touch iq_diCMD *)
END_IF
END_ACTION

ACTION SignalUnSuccessfulExecution:
IF fbLoggerPoint.etLogLevel >= APL.ET_LogLevel.StatusMessage THEN
	fbLoggerPoint.AddLogEntry(	i_etLogLevel	:= APL.ET_LogLevel.StatusMessage,
								i_etDiag		:= GD.ET_Diag.Ok,
								i_udiDiagExt	:= ET_DiagExtExampleLeafModule.Ok,
								i_sMessage		:= Standard.CONCAT(Standard.CONCAT(Standard.CONCAT('Command failed: ', FC_etExampleLeafModuleCmdToString(i_diCmd := iq_stStandardModuleItf.iq_diCmd)),' number: '),DINT_TO_STRING(iq_stStandardModuleItf.iq_diCmd)),
								q_etDiag		:= ,
								q_etDiagExt		:= );
END_IF

iq_stStandardModuleItf.q_xCMDActive := FALSE;
iq_stStandardModuleItf.q_xCMDDone := FALSE;
IF(iq_stStandardModuleItf.iq_diCMD = iq_stStandardModuleItf.q_diCMDActive) THEN
	iq_stStandardModuleItf.iq_diCMD := - iq_stStandardModuleItf.iq_diCMD;
(* ELSE don't touch iq_diCMD *)
END_IF
END_ACTION

END_FUNCTION_BLOCK

// LMC_PacDrive/Application/FC_EtExampleLeafModuleCmdToString
FUNCTION FC_EtExampleLeafModuleCmdToString : STRING[15]
VAR_INPUT
	i_diCmd		: DINT;
END_VAR
VAR_OUTPUT
	q_etDiag	: GD.ET_Diag := GD.ET_Diag.Ok;
	q_etDiagExt	: ET_DiagExtExampleLeafModule := ET_DiagExtExampleLeafModule.Ok;
END_VAR

CASE i_diCMD OF
	ET_ExampleLeafModuleCmd.Homing:
		FC_EtExampleLeafModuleCmdToString := 'Homing';
	ET_ExampleLeafModuleCmd.Auto:
		FC_EtExampleLeafModuleCmdToString := 'Auto';
	ET_ExampleLeafModuleCmd.Stop:
		FC_EtExampleLeafModuleCmdToString := 'Stop';
	ET_ExampleLeafModuleCmd.Start:
		FC_EtExampleLeafModuleCmdToString := 'Start';
	ET_ExampleLeafModuleCmd.Hold:
		FC_EtExampleLeafModuleCmdToString := 'Hold';
	ELSE
		FC_EtExampleLeafModuleCmdToString := CONCAT('Unkown Cmd ', DINT_TO_STRING(i_diCMD));
		
		q_etDiag := GD.ET_Diag.InputParameterInvalid;
		q_etDiagExt := ET_DiagExtExampleLeafModule.UnknownCmd;
END_CASE

END_FUNCTION

// LMC_PacDrive/Application/FC_EtExampleLeafModuleStateToString
FUNCTION FC_EtExampleLeafModuleStateToString : STRING[25]
VAR_INPUT
	i_etState	: ET_ExampleLeafModuleState;
END_VAR
VAR_OUTPUT
	q_etDiag	: GD.ET_Diag := GD.ET_Diag.Ok;
	q_etDiagExt	: ET_DiagExtExampleLeafModule := ET_DiagExtExampleLeafModule.Ok;
END_VAR

CASE i_etState OF
	ET_ExampleLeafModuleState.Disabled:
		FC_EtExampleLeafModuleStateToString := 'Disabled';
	ET_ExampleLeafModuleState.Initializing:
		FC_EtExampleLeafModuleStateToString := 'Initializing';
	ET_ExampleLeafModuleState.NoOp:
		FC_EtExampleLeafModuleStateToString := 'NoOp';
	ET_ExampleLeafModuleState.HomingWaitForStart:
		FC_EtExampleLeafModuleStateToString := 'HomingWaitForStart';
	ET_ExampleLeafModuleState.HomingExecuting:
		FC_EtExampleLeafModuleStateToString := 'HomingExecuting';
	ET_ExampleLeafModuleState.HomingDone:
		FC_EtExampleLeafModuleStateToString := 'HomingDone';
	ET_ExampleLeafModuleState.AutoWaitForStart:
		FC_EtExampleLeafModuleStateToString := 'AutoWaitForStart';
	ET_ExampleLeafModuleState.AutoRunning:
		FC_EtExampleLeafModuleStateToString := 'AutoRunning';
	ELSE
		FC_EtExampleLeafModuleStateToString := CONCAT('Unkown State ', UDINT_TO_STRING(i_etState));
		
		q_etDiag := GD.ET_Diag.InputParameterInvalid;
		q_etDiagExt := ET_DiagExtExampleLeafModule.UnknownState;
END_CASE

END_FUNCTION

// LMC_PacDrive/Application/FC_EtDiagExtExampleLeafModuleToString
FUNCTION FC_EtDiagExtExampleLeafModuleToString : STRING[80]

VAR_INPUT
	i_etDiagExt : ET_DiagExtExampleLeafModule;
END_VAR

VAR_OUTPUT
	q_etDiag	: GD.ET_Diag := GD.ET_Diag.Ok;
	q_etDiagExt	: ET_DiagExtExampleLeafModule := ET_DiagExtExampleLeafModule.Ok;
END_VAR

VAR
END_VAR

CASE i_etDiagExt OF
	ET_DiagExtExampleLeafModule.Ok:										FC_EtDiagExtExampleLeafModuleToString := 'Ok';
	ET_DiagExtExampleLeafModule.Disabled:								FC_EtDiagExtExampleLeafModuleToString := 'Disabled';
	ET_DiagExtExampleLeafModule.Initializing:							FC_EtDiagExtExampleLeafModuleToString := 'Initializing';
	ET_DiagExtExampleLeafModule.NoOp:									FC_EtDiagExtExampleLeafModuleToString := 'NoOp';
	ET_DiagExtExampleLeafModule.HomingWaitForStart:						FC_EtDiagExtExampleLeafModuleToString := 'HomingWaitForStart';
	ET_DiagExtExampleLeafModule.HomingExecuting:						FC_EtDiagExtExampleLeafModuleToString := 'HomingExecuting';
	ET_DiagExtExampleLeafModule.HomingDone:								FC_EtDiagExtExampleLeafModuleToString := 'HomingDone';
	ET_DiagExtExampleLeafModule.AutoWaitForStart:						FC_EtDiagExtExampleLeafModuleToString := 'AutoWaitForStart';
	ET_DiagExtExampleLeafModule.AutoRunning:							FC_EtDiagExtExampleLeafModuleToString := 'AutoRunning';
	ET_DiagExtExampleLeafModule.Working:								FC_EtDiagExtExampleLeafModuleToString := 'Working';

	ET_DiagExtExampleLeafModule.UnknownDiagExtExampleLeafModule:		FC_EtDiagExtExampleLeafModuleToString := 'UnknownDiagExtExampleLeafModule';
	ET_DiagExtExampleLeafModule.SubModuleAddInterfacesInvalidPointer:	FC_EtDiagExtExampleLeafModuleToString := 'SubModuleAddInterfacesInvalidPointer';
	ET_DiagExtExampleLeafModule.SubModuleConstantRange:					FC_EtDiagExtExampleLeafModuleToString := 'SubModuleConstantRange';
	ET_DiagExtExampleLeafModule.MissingExtInit:							FC_EtDiagExtExampleLeafModuleToString := 'MissingExtInit';
	ET_DiagExtExampleLeafModule.ReactionOffsetRange:					FC_EtDiagExtExampleLeafModuleToString := 'ReactionOffsetRange';
	ET_DiagExtExampleLeafModule.DriveInvalid:							FC_EtDiagExtExampleLeafModuleToString := 'DriveInvalid';
	
	ET_DiagExtExampleLeafModule.CmdUnknown:								FC_EtDiagExtExampleLeafModuleToString := 'CmdUnknown';
	ET_DiagExtExampleLeafModule.CmdImpossibleOverwrite:					FC_EtDiagExtExampleLeafModuleToString := 'CmdImpossibleOverwrite';
	ET_DiagExtExampleLeafModule.CmdImpossibleState:						FC_EtDiagExtExampleLeafModuleToString := 'CmdImpossibleState';
	ET_DiagExtExampleLeafModule.CmdImpossibleReaction:					FC_EtDiagExtExampleLeafModuleToString := 'CmdImpossibleReaction';
	
	ET_DiagExtExampleLeafModule.AsyncStop:								FC_EtDiagExtExampleLeafModuleToString := 'AsyncStop';
	ET_DiagExtExampleLeafModule.SyncStopEL:								FC_EtDiagExtExampleLeafModuleToString := 'SyncStopEL';
	ET_DiagExtExampleLeafModule.SyncStopEH:								FC_EtDiagExtExampleLeafModuleToString := 'SyncStopEH';
	ET_DiagExtExampleLeafModule.StopEndOfCycle:							FC_EtDiagExtExampleLeafModuleToString := 'StopEndOfCycle';
	
	ET_DiagExtExampleLeafModule.DriveFatalException:					FC_EtDiagExtExampleLeafModuleToString := 'DriveFatalException';
	ET_DiagExtExampleLeafModule.DriveException:							FC_EtDiagExtExampleLeafModuleToString := 'DriveException';
	ET_DiagExtExampleLeafModule.DriveWarning:							FC_EtDiagExtExampleLeafModuleToString := 'DriveWarning';
	
	ET_DiagExtExampleLeafModule.UnknownState:							FC_EtDiagExtExampleLeafModuleToString := 'UnknownState';
	ET_DiagExtExampleLeafModule.UnknownCmd:								FC_EtDiagExtExampleLeafModuleToString := 'UnknownCmd';
	ET_DiagExtExampleLeafModule.RandomException:						FC_EtDiagExtExampleLeafModuleToString := 'RandomException';

	ET_DiagExtExampleLeafModule.CurrentStandardItfInvalidPointer:		FC_EtDiagExtExampleLeafModuleToString := 'CurrentStandardItfInvalidPointer';
	ET_DiagExtExampleLeafModule.CurrentAddItfInvalidPointer:			FC_EtDiagExtExampleLeafModuleToString := 'CurrentAddItfInvalidPointer';
	
	ET_DiagExtExampleLeafModule.ParentInvalid:							FC_EtDiagExtExampleLeafModuleToString := 'ParentInvalid';
	ET_DiagExtExampleLeafModule.ParentNotRegistered:					FC_EtDiagExtExampleLeafModuleToString := 'ParentNotRegistered';
	ET_DiagExtExampleLeafModule.MaxNumberOfLoggerPointsExeeded:			FC_EtDiagExtExampleLeafModuleToString := 'MaxNumberOfLoggerPointsExeeded';
	ET_DiagExtExampleLeafModule.UnexpectedDiagExt:						FC_EtDiagExtExampleLeafModuleToString := 'UnexpectedDiagExt';
	
	ELSE
		FC_EtDiagExtExampleLeafModuleToString := Standard.CONCAT('Unkown ET_DiagExtExampleLeafModule ', UDINT_TO_STRING(i_etDiagExt));
		
		q_etDiag	:= GD.ET_Diag.InputParameterInvalid;
		q_etDiagExt	:= ET_DiagExtExampleLeafModule.UnknownDiagExtExampleLeafModule;
END_CASE

END_FUNCTION

// LMC_PacDrive/Application/FB_ExampleLeafModuleController
FUNCTION_BLOCK FB_ExampleLeafModuleController

VAR_INPUT
	i_xEnable				: BOOL;
END_VAR

VAR_IN_OUT
	iq_stStandardModuleItf	: TPL.ST_StandardModuleInterface;
	iq_stStandardMotionItf	: TPL.ST_StandardMotionInterface;
	iq_stExceptionList		: TPL.ST_ExceptionList;
	iq_stLogDataList		: TPL.ST_LogDataList;
END_VAR

VAR_OUTPUT
	q_xActive				: BOOL;
	q_xReady				: BOOL;
	q_etDiag				: GD.ET_Diag := GD.ET_Diag.Ok;
	q_etDiagExt				: ET_DiagExtExampleLeafModule := ET_DiagExtExampleLeafModule.Disabled;
	q_sMsg					: STRING[80] := '';
END_VAR

VAR
	xEnableFlag				: BOOL;
	udiTmp					: UDINT;
END_VAR

IF i_xEnable AND NOT xEnableFlag THEN
	xEnableFlag	:= TRUE;
	
	q_xActive	:= TRUE;

	q_etDiag	:= GD.ET_Diag.Ok;
	q_etDiagExt := ET_DiagExtExampleLeafModule.Initializing;
	q_sMsg		:= '';
	
	IF ((iq_stStandardModuleItf.iq_stExt.udiNumberOfSubModules <> 0) AND 
	   ((iq_stStandardModuleItf.iq_stExt.pdwSubModulesAddItf = 0) OR (iq_stStandardModuleItf.iq_stExt.dwSubModulesItf = 0))) THEN
	   
		q_etDiag	:= GD.ET_Diag.ExecutionAborted;
		q_etDiagExt	:= ET_DiagExtExampleLeafModule.MissingExtInit;
		q_sMsg		:= 'Missing call of FC_UpdateExampleLeafModuleAddInterfaceStruct';

		RETURN;
	END_IF
	
	udiTmp := ET_ExceptionSource.ExampleLeafModule;
	
	q_xReady := TPL.FC_CheckSubModuleList(	i_dwModuleType		:= UDINT_TO_DWORD(ET_ModuleType.ExampleLeafModule),
											i_udiModuleId		:= iq_stStandardModuleItf.i_udiModuleId,
											i_sModuleName		:= iq_stStandardModuleItf.i_sModuleName,
											i_etSource			:= udiTmp (* Hack around compiler restrictions *),
											iq_stExt			:= iq_stStandardModuleItf.iq_stExt,
											iq_stExceptionList	:= iq_stExceptionList,
											iq_stLogDataList	:= iq_stLogDataList);
											
	IF NOT q_xReady THEN
		xEnableFlag := FALSE;
	END_IF

ELSIF NOT i_xEnable AND xEnableFlag THEN
	xEnableFlag	:= FALSE;
	
	(* No actions required, this simple module does not support jogging or any other things the XXXModuleController would have to handle *)
	q_xReady 	:= FALSE;
	q_xActive	:= FALSE;
	
	q_etDiag	:= GD.ET_Diag.Ok;
	q_etDiagExt	:= ET_DiagExtExampleLeafModule.Disabled;
	q_sMsg		:= '';
END_IF



IF q_xActive AND q_xReady THEN
	(* No actions required, this simple module does not support jogging or any other things the XXXModuleController would have to handle *)
	q_etDiag	:= GD.ET_Diag.Ok;
	q_etDiagExt := ET_DiagExtExampleLeafModule.Working;
	q_sMsg		:= '';
END_IF

END_FUNCTION_BLOCK

// LMC_PacDrive/Application/FC_UpdateExampleLeafModuleAddInterfaceStruct
FUNCTION FC_UpdateExampleLeafModuleAddInterfaceStruct : BOOL

VAR_INPUT
	i_pdwSubModuleAddInterfaces		: POINTER TO DWORD;
	i_udiSubModuleConstant			: UDINT;
END_VAR

VAR_OUTPUT
	q_etDiag						: GD.ET_Diag := GD.ET_Diag.Ok;
	q_etDiagExt						: ET_DiagExtExampleLeafModule := ET_DiagExtExampleLeafModule.Ok;
	q_sMsg							: STRING[80] := '';
END_VAR

VAR_IN_OUT
	iq_stExampleLeafModuleInterface	: ST_ExampleLeafModuleInterface;
END_VAR

VAR
	pdwArrayPos						: POINTER TO DWORD;
END_VAR

IF i_pdwSubModuleAddInterfaces = 0 THEN
	q_etDiag	:= GD.ET_Diag.InputParameterInvalid;
	q_etDiagExt	:= ET_DiagExtExampleLeafModule.SubModuleAddInterfacesInvalidPointer;
	q_sMsg		:= '';
ELSIF i_udiSubModuleConstant < 1 THEN
	q_etDiag	:= GD.ET_Diag.InputParameterInvalid;
	q_etDiagExt := ET_DiagExtExampleLeafModule.SubModuleConstantRange;
	q_sMsg		:= '1 <= i_udiSubModuleConstant';
ELSE
	pdwArrayPos := i_pdwSubModuleAddInterfaces + UDINT_TO_DWORD((i_udiSubModuleConstant-1) * SIZEOF(pdwArrayPos^));
	pdwArrayPos^ := ADR(iq_stExampleLeafModuleInterface);
END_IF

END_FUNCTION

// LMC_PacDrive/Application/SR_NodeWithoutMotionModule
PROGRAM SR_NodeWithoutMotionModule

VAR CONSTANT
	(* Standard related constants *)
	c_udiNumberOfGroups			: UDINT := 0;			(* Maximum number of groups *)
	c_udiNumberOfGroupMembers	: UDINT := 0;			(* Maximum number of members per group *)

	c_udiNumberOfCmdTables		: UDINT := 8;			(* Must be the exact number of used CMDTables! *)
	c_udiNumberOfCmdSteps		: UDINT := 16;			(* Make sure that the number of commands/ Steps  that each table
														   contains does not exceed the c_diNumberOfCMDSteps variable.*)

(* System generated code, could be modified for your application *)
	c_udiNumberOfSubModules		: UDINT := 0;				(* Number of SubModules *)
(* End of system generated code, could be modified for your application *)
END_VAR

VAR (*User specific variables*)
	
END_VAR

VAR_IN_OUT
(* TPL.ST_StandardModuleInterface *)	
	iq_stStandardModuleItf			: TPL.ST_StandardModuleInterface;
	
(* ExceptionHandling and Logging *)	
	iq_stExceptionList				: TPL.ST_ExceptionList;
	iq_stLogDataList				: TPL.ST_LogDataList;
END_VAR

VAR
	xInitSuccessful : BOOL := TRUE;
	
	(* Standard related variables *)
	astSubModuleInterface			: ARRAY[1..c_udiNumberOfSubModules] OF TPL.ST_StandardModuleInterface;		(* Interface to modules *)
	aaudiSubModuleGroups			: ARRAY[1..c_udiNumberOfGroups,1..c_udiNumberOfGroupMembers] OF UDINT;
	adwSubModuleAddInterfaces		: ARRAY[1..c_udiNumberOfSubModules] OF DWORD;

	(* Modules related variables *)
	fbModuleController				: TPL.FB_ModuleController;
	etDiagModuleController			: GD.ET_Diag;
	etDiagExtModuleController		: TPL.ET_DiagExt;
	sMsgModuleController			: STRING[80];
	xWaitForStartStep				: BOOL;
	
	astListOfCmdTables				: ARRAY [1..c_udiNumberOfCmdTables] OF TPL.ST_CmdTable;
	udiTableIndex					: UDINT;
	udiStepIndex					: UDINT;
	diStep							: DINT;

	astPrepareTable					: ARRAY [1..c_udiNumberOfCmdSteps] OF TPL.ST_Cmd;		(* Relating  Cmd table *)
	astAutoTable					: ARRAY [1..c_udiNumberOfCmdSteps] OF TPL.ST_Cmd;		(* Relating  Cmd table *)
	astManualTable					: ARRAY [1..c_udiNumberOfCmdSteps] OF TPL.ST_Cmd;		(* Relating  Cmd table *)
	astHoldTable					: ARRAY [1..c_udiNumberOfCmdSteps] OF TPL.ST_Cmd;		(* Relating  Cmd table *)
	astStartTable					: ARRAY [1..c_udiNumberOfCmdSteps] OF TPL.ST_Cmd;		(* Relating  Cmd table *)
	astStopTable					: ARRAY [1..c_udiNumberOfCmdSteps] OF TPL.ST_Cmd;		(* Relating  Cmd table *)
	astBrakeReleaseTable			: ARRAY [1..c_udiNumberOfCmdSteps] OF TPL.ST_Cmd;		(* Relating  Cmd table *)
	astAbortTable					: ARRAY [1..c_udiNumberOfCmdSteps] OF TPL.ST_Cmd;		(* Relating  Cmd table *)

(* ExceptionHandling related variables *)
	fbExceptionHandler				: TPL.FB_ExceptionHandler2;

	aetReactionTranslationMode		: ARRAY[1..c_udiNumberOfSubModules] OF TPL.ET_ReactionTranslationMode;
	aastReactionTranslationTable	: ARRAY[1..c_udiNumberOfSubModules,1..TPL.Gc_udiMaxNumberOfReactions] OF TPL.ST_Reaction;
	astReactionTranslationJobs		: ARRAY[1..c_udiNumberOfSubModules] OF TPL.ST_ReactionTranslationJobs;
	
(* Exception declaration *)
	stUserException1				: TPL.ST_Exception;
	stUserException2				: TPL.ST_Exception;
	xModuleUserException1			: BOOL;
	xModuleUserException2			: BOOL;
	
	stUpdateStructsException		: TPL.ST_Exception;
	xUpdateStructsException			: BOOL;
	
	stInitReactionsException		: TPL.ST_Exception;
	xInitReactionsException			: BOOL;
	
	stInitSubModulesException		: TPL.ST_Exception;
	xInitSubModulesException		: BOOL;

(* Logging related variables*)
	fbLogger						: TPL.FB_Logger;
	fbLoggerPoint					: APL.FB_LoggerPoint;

(* OnlineChange related variables *)
	fbDetectOnlineChange			: TPL.FB_DetectOnlineChange;
	xDetectOnlineChangeActive		: BOOL; 
	xDetectOnlineChangeReady		: BOOL; 
	etDetectOnlineChangeDiag		: GD.ET_Diag;
	etDetectOnlineChangeDiagExt		: TPL.ET_DiagExt; 
	sDetectOnlineChangeMsg			: STRING[80];
	
(* POU-Feedback related variables*)	
	etDiag			: GD.ET_Diag;
	etDiagExtTPL	: TPL.ET_DiagExt;
	etDiagExtAXM	: AXM.ET_DiagExt;
END_VAR

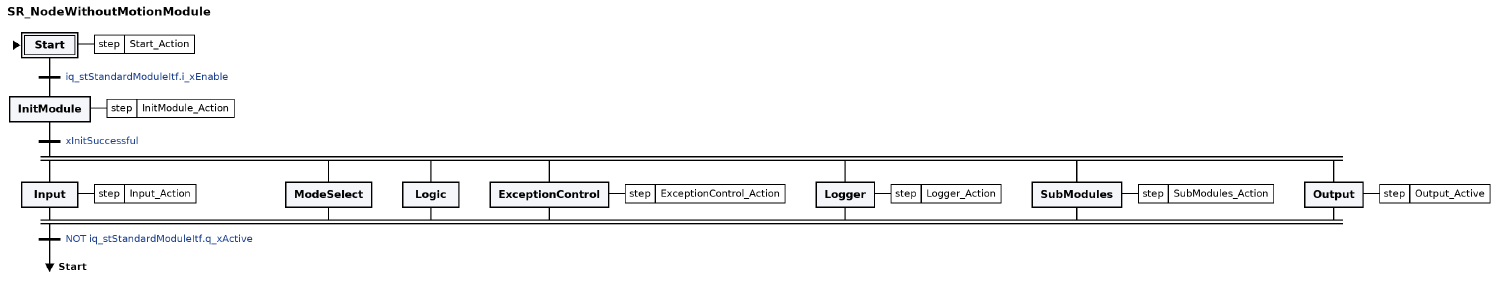
INITIAL_STEP Start:
    Start_Action(N);  // step action
END_STEP
TRANSITION FROM Start TO InitModule
    := iq_stStandardModuleItf.i_xEnable;
END_TRANSITION
STEP InitModule:
    InitModule_Action(N);  // step action
END_STEP
TRANSITION FROM InitModule TO (Input, ModeSelect, Logic, ExceptionControl, Logger, SubModules, Output)
    := xInitSuccessful;
END_TRANSITION
STEP Input:
    Input_Action(N);  // step action
END_STEP
STEP ModeSelect:
END_STEP
STEP Logic:
END_STEP
STEP ExceptionControl:
    ExceptionControl_Action(N);  // step action
END_STEP
STEP Logger:
    Logger_Action(N);  // step action
END_STEP
STEP SubModules:
    SubModules_Action(N);  // step action
END_STEP
STEP Output:
    Output_Active(N);  // step action
END_STEP
TRANSITION FROM (Input, ModeSelect, Logic, ExceptionControl, Logger, SubModules, Output) TO Start
    := NOT iq_stStandardModuleItf.q_xActive;
END_TRANSITION

ACTION ExceptionControl_Action:
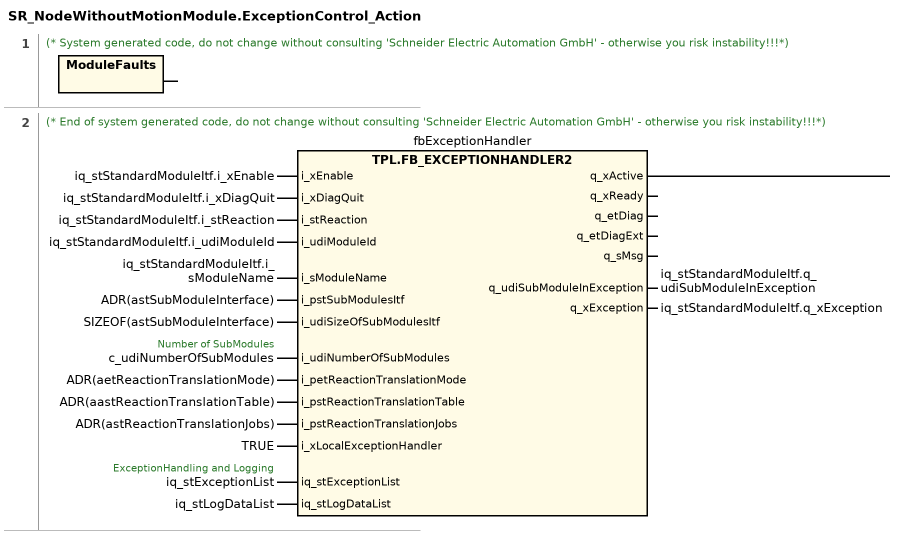
// NETWORK 1
// (* System generated code, do not change without consulting 'Schneider Electric Automation GmbH' - otherwise you risk instability!!!*)
ModuleFaults();

// NETWORK 2
// (* End of system generated code, do not change without consulting 'Schneider Electric Automation GmbH' - otherwise you risk instability!!!*)
//   fbExceptionHandler: ExceptionHandling related variables
//   c_udiNumberOfSubModules: Number of SubModules
//   iq_stExceptionList: ExceptionHandling and Logging
fbExceptionHandler(
    i_xEnable := iq_stStandardModuleItf.i_xEnable,
    i_xDiagQuit := iq_stStandardModuleItf.i_xDiagQuit,
    i_stReaction := iq_stStandardModuleItf.i_stReaction,
    i_udiModuleId := iq_stStandardModuleItf.i_udiModuleId,
    i_sModuleName := iq_stStandardModuleItf.i_sModuleName,
    i_pstSubModulesItf := ADR(astSubModuleInterface),
    i_udiSizeOfSubModulesItf := SIZEOF(astSubModuleInterface),
    i_udiNumberOfSubModules := c_udiNumberOfSubModules,
    i_petReactionTranslationMode := ADR(aetReactionTranslationMode),
    i_pstReactionTranslationTable := ADR(aastReactionTranslationTable),
    i_pstReactionTranslationJobs := ADR(astReactionTranslationJobs),
    i_xLocalExceptionHandler := TRUE,
    iq_stExceptionList := iq_stExceptionList,
    iq_stLogDataList := iq_stLogDataList,
    q_udiSubModuleInException => iq_stStandardModuleItf.q_udiSubModuleInException,
    q_xException => iq_stStandardModuleItf.q_xException); // TPL.FB_EXCEPTIONHANDLER2
END_ACTION

ACTION Init_CmdTables:
(* System generated code, could be modified for your application *)

(*********************************************************************************************************************)
(*** Prepare  ***)

TPL.FC_FirstLastStepEmptyTable(udiStepIndex, diStep);
astPrepareTable[udiStepIndex].sTitle					:= 'End';
astPrepareTable[udiStepIndex].udiModuleName				:= 0;
astPrepareTable[udiStepIndex].diStep					:= diStep;
astPrepareTable[udiStepIndex].diCMD						:= 0;
astPrepareTable[udiStepIndex].timTimeOut				:= T#0MS;
astPrepareTable[udiStepIndex].xEndCMD					:= TRUE;

TPL.FC_FirstCmdTable(iq_udiTableIndex:= udiTableIndex);
astListofCMDTables[udiTableIndex].sTitle				:= 'Prepare';
astListofCMDTables[udiTableIndex].diCMD					:= ET_Cmd.Prepare;
astListofCMDTables[udiTableIndex].udiNumberOfCmdSteps	:= udiStepIndex;

(*********************************************************************************************************************)
(*** Auto  ***)

TPL.FC_FirstLastStepEmptyTable(udiStepIndex, diStep);
astAutoTable[udiStepIndex].sTitle						:= 'End';
astAutoTable[udiStepIndex].udiModuleName				:= 0;
astAutoTable[udiStepIndex].diStep						:= diStep;
astAutoTable[udiStepIndex].diCMD						:= 0;
astAutoTable[udiStepIndex].timTimeOut					:= T#0MS;
astAutoTable[udiStepIndex].xEndCMD						:= TRUE;

TPL.FC_NextCmdTable(iq_udiTableIndex:= udiTableIndex);
astListofCMDTables[udiTableIndex].sTitle				:= 'Auto';
astListofCMDTables[udiTableIndex].diCMD					:= ET_Cmd.Auto;
astListofCMDTables[udiTableIndex].udiNumberOfCmdSteps	:= udiStepIndex;

(*********************************************************************************************************************)
(*** Manual  ***)

TPL.FC_FirstLastStepEmptyTable(udiStepIndex, diStep);
astManualTable[udiStepIndex].sTitle						:= 'End';
astManualTable[udiStepIndex].udiModuleName				:= 0;
astManualTable[udiStepIndex].diStep						:= diStep;
astManualTable[udiStepIndex].diCMD						:= 0;
astManualTable[udiStepIndex].timTimeOut					:= T#0MS;
astManualTable[udiStepIndex].xEndCMD					:= TRUE;

TPL.FC_NextCmdTable(iq_udiTableIndex:= udiTableIndex);
astListofCMDTables[udiTableIndex].sTitle				:= 'Manual';
astListofCMDTables[udiTableIndex].diCMD					:= ET_Cmd.Manual;
astListofCMDTables[udiTableIndex].udiNumberOfCmdSteps	:= udiStepIndex;

(*********************************************************************************************************************)
(*** Stop ***)

TPL.FC_FirstLastStepEmptyTable(udiStepIndex, diStep);
astStopTable[udiStepIndex].sTitle						:= 'End';
astStopTable[udiStepIndex].udiModuleName				:= 0;
astStopTable[udiStepIndex].diStep						:= diStep;
astStopTable[udiStepIndex].diCMD						:= 0;
astStopTable[udiStepIndex].timTimeOut					:= T#0MS;
astStopTable[udiStepIndex].xEndCMD						:= TRUE;

TPL.FC_NextCmdTable(iq_udiTableIndex:= udiTableIndex);
astListofCMDTables[udiTableIndex].sTitle				:= 'Stop';
astListofCMDTables[udiTableIndex].diCMD					:= ET_Cmd.Stop;
astListofCMDTables[udiTableIndex].udiNumberOfCmdSteps	:= udiStepIndex;

(*********************************************************************************************************************)
(*** Start ***)

TPL.FC_FirstLastStepEmptyTable(udiStepIndex, diStep);
astStartTable[udiStepIndex].sTitle						:= 'End';
astStartTable[udiStepIndex].udiModuleName				:= 0;
astStartTable[udiStepIndex].diStep						:= diStep;
astStartTable[udiStepIndex].diCMD						:= 0;
astStartTable[udiStepIndex].timTimeOut					:= T#0MS;
astStartTable[udiStepIndex].xEndCMD						:= TRUE;

TPL.FC_NextCmdTable(iq_udiTableIndex:= udiTableIndex);
astListofCMDTables[udiTableIndex].sTitle				:= 'Start';
astListofCMDTables[udiTableIndex].diCMD					:= ET_Cmd.Start;
astListofCMDTables[udiTableIndex].udiNumberOfCmdSteps	:= udiStepIndex;

(*********************************************************************************************************************)
(*** Abort ***)

TPL.FC_FirstLastStepEmptyTable(udiStepIndex, diStep);
astAbortTable[udiStepIndex].sTitle						:= 'End';
astAbortTable[udiStepIndex].udiModuleName				:= 0;
astAbortTable[udiStepIndex].diStep						:= diStep;
astAbortTable[udiStepIndex].diCMD						:= 0;
astAbortTable[udiStepIndex].timTimeOut					:= T#0MS;
astAbortTable[udiStepIndex].xEndCMD						:= TRUE;

TPL.FC_NextCmdTable(iq_udiTableIndex:= udiTableIndex);
astListofCMDTables[udiTableIndex].sTitle				:= 'Abort';
astListofCMDTables[udiTableIndex].diCMD					:= ET_Cmd.Abort;
astListofCMDTables[udiTableIndex].udiNumberOfCmdSteps	:= udiStepIndex;

(*********************************************************************************************************************)
(*** Hold ***)

TPL.FC_FirstLastStepEmptyTable(udiStepIndex, diStep);
astHoldTable[udiStepIndex].sTitle						:= 'End';
astHoldTable[udiStepIndex].udiModuleName				:= 0;
astHoldTable[udiStepIndex].diStep						:= diStep;
astHoldTable[udiStepIndex].diCMD						:= 0;
astHoldTable[udiStepIndex].timTimeOut					:= T#0MS;
astHoldTable[udiStepIndex].xEndCMD						:= TRUE;

TPL.FC_NextCmdTable(iq_udiTableIndex:= udiTableIndex);
astListofCMDTables[udiTableIndex].sTitle				:= 'Hold';
astListofCMDTables[udiTableIndex].diCMD					:= ET_Cmd.Hold;
astListofCMDTables[udiTableIndex].udiNumberOfCmdSteps	:= udiStepIndex;

(*********************************************************************************************************************)
(*** Brake Release ***)

TPL.FC_FirstLastStepEmptyTable(udiStepIndex, diStep);
astBrakeReleaseTable[udiStepIndex].sTitle				:= 'End';
astBrakeReleaseTable[udiStepIndex].udiModuleName		:= 0;
astBrakeReleaseTable[udiStepIndex].diStep				:= diStep;
astBrakeReleaseTable[udiStepIndex].diCMD				:= 0;
astBrakeReleaseTable[udiStepIndex].timTimeOut			:= T#0MS;
astBrakeReleaseTable[udiStepIndex].xEndCMD				:= TRUE;

TPL.FC_NextCmdTable(iq_udiTableIndex:= udiTableIndex);
astListofCMDTables[udiTableIndex].sTitle				:= 'Brake Release';
astListofCMDTables[udiTableIndex].diCMD					:= ET_Cmd.BrakeRelease;
astListofCMDTables[udiTableIndex].udiNumberOfCmdSteps	:= udiStepIndex;

(* End of system generated code, could be modified for your application *)
END_ACTION

ACTION Init_Exceptions:
(* System generated code, could be modified for your application *)
stUpdateStructsException.etDiag												:= GD.ET_Diag.UnexpectedProgramBehavior;
stUpdateStructsException.udiDiagExt											:= ET_DiagExt.UpdateStructsException;
stUpdateStructsException.sDiagExt											:= FC_EtDiagExtToString(i_etDiagExt := stUpdateStructsException.udiDiagExt);
stUpdateStructsException.sMsg												:= '';	(* Replaced on usage *)
stUpdateStructsException.udiModuleId										:= iq_stStandardModuleItf.i_udiModuleId;
stUpdateStructsException.sModuleName										:= iq_stStandardModuleItf.i_sModuleName;
stUpdateStructsException.stReaction.axReaction[TPL.ET_Reaction.AsyncStop]	:= TRUE;
stUpdateStructsException.etSource											:= TPL.ET_ExceptionSource.NodeModule;
stUpdateStructsException.timDelayTime										:= T#0MS;
stUpdateStructsException.wHmiAttributes										:= 0;
stUpdateStructsException.xAutoQuit											:= FALSE;

stInitReactionsException.etDiag												:= GD.ET_Diag.UnexpectedProgramBehavior;
stInitReactionsException.udiDiagExt											:= ET_DiagExt.InitReactionsException;
stInitReactionsException.sDiagExt											:= FC_EtDiagExtToString(i_etDiagExt := stInitReactionsException.udiDiagExt);
stInitReactionsException.sMsg												:= '';	(* Replaced on usage *)
stInitReactionsException.udiModuleId										:= iq_stStandardModuleItf.i_udiModuleId;
stInitReactionsException.sModuleName										:= iq_stStandardModuleItf.i_sModuleName;
stInitReactionsException.stReaction.axReaction[TPL.ET_Reaction.AsyncStop]	:= TRUE;
stInitReactionsException.etSource											:= TPL.ET_ExceptionSource.NodeModule;
stInitReactionsException.timDelayTime										:= T#0MS;
stInitReactionsException.wHmiAttributes										:= 0;
stInitReactionsException.xAutoQuit											:= FALSE;

stInitSubModulesException.etDiag											:= GD.ET_Diag.UnexpectedProgramBehavior;
stInitSubModulesException.udiDiagExt										:= ET_DiagExt.InitSubModulesException;
stInitSubModulesException.sDiagExt											:= FC_EtDiagExtToString(i_etDiagExt := stInitSubModulesException.udiDiagExt);
stInitSubModulesException.sMsg												:= '';	(* Replaced on usage *)
stInitSubModulesException.udiModuleId										:= iq_stStandardModuleItf.i_udiModuleId;
stInitSubModulesException.sModuleName										:= iq_stStandardModuleItf.i_sModuleName;
stInitSubModulesException.stReaction.axReaction[TPL.ET_Reaction.AsyncStop]	:= TRUE;
stInitSubModulesException.etSource											:= TPL.ET_ExceptionSource.NodeModule;
stInitSubModulesException.timDelayTime										:= T#0MS;
stInitSubModulesException.wHmiAttributes									:= 0;
stInitSubModulesException.xAutoQuit											:= FALSE;


(*------------------------------------------------------------------------------------------*)
(* Init User Exceptions *)

	// TPL.ET_Reaction.AsyncStop
	// TPL.ET_Reaction.SyncStopEL
	// TPL.ET_Reaction.SyncStopEH
	// TPL.ET_Reaction.StopEndOfCycle
	// TPL.ET_Reaction.MainsContactorOff

(*------------------------------------------------------------------------------------------*)
stUserException1.etDiag														:= GD.ET_Diag.ExecutionAborted;
stUserException1.udiDiagExt													:= ET_DiagExtUser.Exception1FromEquipmentModule;
stUserException1.sDiagExt													:= FC_EtDiagExtUserToString(i_etDiagExt := stUserException1.udiDiagExt);
stUserException1.sMsg														:= 'User Exception 1';
stUserException1.udiModuleId												:= iq_stStandardModuleItf.i_udiModuleId;
stUserException1.sModuleName												:= iq_stStandardModuleItf.i_sModuleName;
stUserException1.etSource													:= TPL.ET_ExceptionSource.User;
stUserException1.timDelayTime												:= T#0MS;
stUserException1.wHmiAttributes												:= 0;
stUserException1.xAutoQuit													:= FALSE;
stUserException1.stReaction.axReaction[TPL.Gc_udiUserReactionOffset + 2]	:= TRUE;

stUserException2.etDiag														:= GD.ET_Diag.ExecutionAborted;
stUserException2.udiDiagExt													:= ET_DiagExtUser.Exception2FromEquipmentModule;
stUserException2.sDiagExt													:= FC_EtDiagExtUserToString(i_etDiagExt := stUserException2.udiDiagExt);
stUserException2.sMsg														:= 'User Exception 2';
stUserException2.udiModuleId												:= iq_stStandardModuleItf.i_udiModuleId;
stUserException2.sModuleName												:= iq_stStandardModuleItf.i_sModuleName;
stUserException2.etSource													:= TPL.ET_ExceptionSource.User;
stUserException2.timDelayTime												:= T#0MS;
stUserException2.wHmiAttributes												:= 0;
stUserException2.xAutoQuit													:= FALSE;
stUserException2.stReaction.axReaction[TPL.Gc_udiUserReactionOffset + 2]	:= TRUE;

(* End of system generated code, could be modified for your application *)
END_ACTION

ACTION Init_Reactions:
(* System generated code, only to be changed by experienced programmers *)
IF c_udiNumberOfSubModules < 1 THEN
	RETURN;
END_IF

(* Change of default reactions only on demand *)
(* Compare SR MainMachine Action Init_Reactions *)

xInitReactionsException := FALSE;

(*****************************************************************************************************************************************************)
(* Init ReactionTranslationMode *)

TPL.FC_InitReactionTranslationMode(	i_udiNumberOfSubModules			:= c_udiNumberOfSubModules,
									i_petReactionTranslationMode	:= ADR(aetReactionTranslationMode),
									q_etDiag						=> etDiag,
									q_etDiagExt						=> etDiagExtTPL);
							
IF etDiag <> GD.ET_Diag.Ok AND NOT xInitReactionsException THEN
	xInitReactionsException := TRUE;
	
	stInitReactionsException.sMsg := PDL.FC_MultiConcat(i_sString1 := 'InitReactionTranslationMode - ', 
														i_sString2 := GD.FC_EtDiagToString(i_etDiag := etDiag), 
														i_sString3 := ' - ', 
														i_sString4 := TPL.FC_EtDiagExtToString(i_etDiagExt := etDiagExtTPL));
END_IF	

(*****************************************************************************************************************************************************)
(* Init ReactionTranslationTable *)	

TPL.FC_InitReactionTranslationTable(i_udiNumberOfSubModules			:= c_udiNumberOfSubModules,
									i_pstReactionTranslationTable	:= ADR(aastReactionTranslationTable),
									q_etDiag						=> etDiag,
									q_etDiagExt						=> etDiagExtTPL);
									
IF etDiag <> GD.ET_Diag.Ok AND NOT xInitReactionsException THEN
	xInitReactionsException := TRUE;
	
	stInitReactionsException.sMsg := PDL.FC_MultiConcat(i_sString1 := 'InitReactionTranslationTable - ', 
														i_sString2 := GD.FC_EtDiagToString(i_etDiag := etDiag), 
														i_sString3 := ' - ', 
														i_sString4 := TPL.FC_EtDiagExtToString(i_etDiagExt := etDiagExtTPL));
END_IF		

(*****************************************************************************************************************************************************)
(* Init ReactionTranslationJobs *)	
								
TPL.FC_InitReactionTranslationJobs( i_udiNumberOfSubModules			:= c_udiNumberOfSubModules,
									i_pstReactionTranslationJobs	:= ADR(astReactionTranslationJobs),
									q_etDiag						=> etDiag,
									q_etDiagExt						=> etDiagExtTPL);
						
IF etDiag <> GD.ET_Diag.Ok AND NOT xInitReactionsException THEN
	xInitReactionsException := TRUE;
	
	stInitReactionsException.sMsg := PDL.FC_MultiConcat(i_sString1 := 'InitReactionTranslationJobs - ', 
														i_sString2 := GD.FC_EtDiagToString(i_etDiag := etDiag), 
														i_sString3 := ' - ', 
														i_sString4 := TPL.FC_EtDiagExtToString(i_etDiagExt := etDiagExtTPL));
END_IF		

(*****************************************************************************************************************************************************)
(* Set exception if any exception occurred *)

fbExceptionHandler.SetException(i_xExceptionActive	:= xInitReactionsException, 
								iq_stException		:= stInitReactionsException, 
								iq_stExceptionList	:= iq_stExceptionList);
					
xInitSuccessful := xInitSuccessful AND NOT xInitReactionsException;

etDiag := GD.ET_Diag.Ok;
(* End of system generated code, only to be changed by experienced programmers *)
END_ACTION

ACTION Init_SubModules:
(* System generated code, could be modified for your application *)

(* Module Group declaration *)

(* aaudiSubModuleGroups[c_diNWMGroup1-TPL.Gc_udiGroupOffset,TPL.ET_Group.Member1]	:= 0; *)	(* The c_diMaster is the first element of the group c_diAlphaGroup1 *)
(* aaudiSubModuleGroups[c_diNWMGroup1-TPL.Gc_udiGroupOffset,TPL.ET_Group.Member2]	:= 0; *)	(* There is no second element of the group c_diAlphaGroup1 *)

(* aaudiSubModuleGroups[c_diNWMGroup2-TPL.Gc_udiGroupOffset,TPL.ET_Group.Member1]	:= 0; *)	(* There is no first element of the group c_diAlphaGroup2 *)
(* aaudiSubModuleGroups[c_diNWMGroup2-TPL.Gc_udiGroupOffset,TPL.ET_Group.Member2]	:= 0; *)	(* There is no second element of the group c_diAlphaGroup2 *)

(* End of system generated code, could be modified for your application *)


(* System generated code, do not change without consulting 'Schneider Electric Automation GmbH' - otherwise you risk instability!!!*)
xInitSubModulesException := FALSE;

(*****************************************************************************************************************************************************)
(* Set IDs of SubModules *)	

TPL.FC_SetSubModuleIds(	i_udiMainModuleID			:= iq_stStandardModuleItf.i_udiModuleId,
						i_pstSubModulesItf			:= ADR(astSubModuleInterface),
						i_udiNumberOfSubModules		:= c_udiNumberOfSubModules,
						q_etDiag					=> etDiag,
						q_etDiagExt					=> etDiagExtTPL);
					
IF etDiag <> GD.ET_Diag.Ok AND NOT xInitSubModulesException THEN
	xInitSubModulesException := TRUE;
	
	stInitSubModulesException.sMsg := PDL.FC_MultiConcat(	i_sString1 := 'SetSubModuleIds - ', 
															i_sString2 := GD.FC_EtDiagToString(i_etDiag := etDiag), 
															i_sString3 := ' - ', 
															i_sString4 := TPL.FC_EtDiagExtToString(i_etDiagExt := etDiagExtTPL));
END_IF	

(*****************************************************************************************************************************************************)
(* Set exception if any exception occurred *)

fbExceptionHandler.SetException(i_xExceptionActive	:= xInitSubModulesException, 
								iq_stException		:= stInitSubModulesException, 
								iq_stExceptionList	:= iq_stExceptionList);

xInitSuccessful := xInitSuccessful AND NOT xInitSubModulesException;
					
etDiag := GD.ET_Diag.Ok;
(* End of system generated code, do not change without consulting 'Schneider Electric Automation GmbH' - otherwise you risk instability!!!*)
END_ACTION

ACTION InitModule_Action:
(* This step is used for initialisations after being enabled *)

(* System generated code, could be modified for your application *)
xInitSuccessful := TRUE;

Init_Exceptions();
(* End of system generated code, could be modified for your application *)

(* System generated code, do not change without consulting 'Schneider Electric Automation GmbH' - otherwise you risk instability!!!*)
iq_stStandardModuleItf.q_xActive		:= TRUE;
iq_stStandardModuleItf.q_xReady			:= FALSE;
iq_stStandardModuleItf.q_etDiag			:= GD.ET_Diag.Ok;
iq_stStandardModuleItf.q_udiDiagExt		:= ET_DiagExt.Initializing;
iq_stStandardModuleItf.q_sDiagExt		:= FC_EtDiagExtToString(i_etDiagExt := ET_DiagExt.Initializing);
iq_stStandardModuleItf.q_sMsg			:= '';

Init_SubModules();
Init_CmdTables();
Init_Reactions();
UpdateStructs();
(* End of system generated code, do not change without consulting 'Schneider Electric Automation GmbH' - otherwise you risk instability!!!*)
fbModuleController.RegisterLoggerPoint(	i_ifParent	:= fbLoggerPoint,
										i_sName		:= 'ModuleController',
										q_etDiag	=> ,
										q_etDiagExt	=> );
fbExceptionHandler.RegisterLoggerPoint(	i_ifParent	:= fbLoggerPoint,
										i_sName		:= 'ExceptionHandler',
										q_etDiag	=> ,
										q_etDiagExt	=> );
(* Application specific code *)
(* ToDo: Add your application specific code here *)
;
(* End of application specific code *)
END_ACTION

ACTION Input_Action:
(* System generated code, do not change without consulting 'Schneider Electric Automation GmbH' - otherwise you risk instability!!!*)
UpdateStructs();
(* End of system generated code, do not change without consulting 'Schneider Electric Automation GmbH' - otherwise you risk instability!!!*)
END_ACTION

ACTION Logger_Action:
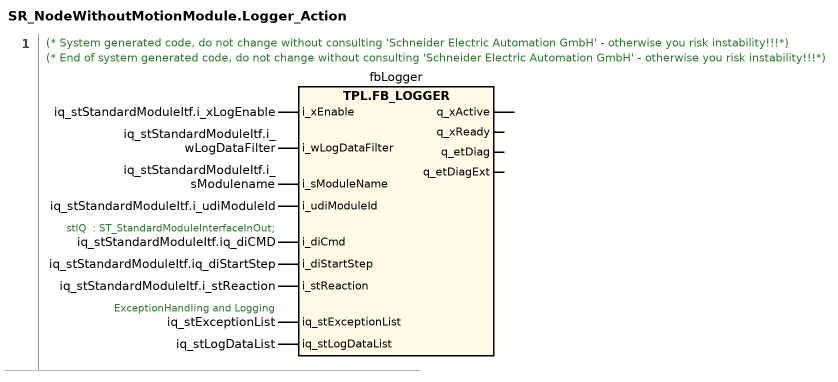
// NETWORK 1
// 					(* System generated code, do not change without consulting 'Schneider Electric Automation GmbH' - otherwise you risk instability!!!*)
// (* End of system generated code, do not change without consulting 'Schneider Electric Automation GmbH' - otherwise you risk instability!!!*)
//
//   fbLogger: Logging related variables
//   iq_stStandardModuleItf.iq_diCMD: stIQ : ST_StandardModuleInterfaceInOut;
//   iq_stExceptionList: ExceptionHandling and Logging
fbLogger(
    i_xEnable := iq_stStandardModuleItf.i_xLogEnable,
    i_wLogDataFilter := iq_stStandardModuleItf.i_wLogDataFilter,
    i_sModuleName := iq_stStandardModuleItf.i_sModulename,
    i_udiModuleId := iq_stStandardModuleItf.i_udiModuleId,
    i_diCmd := iq_stStandardModuleItf.iq_diCMD,
    i_diStartStep := iq_stStandardModuleItf.iq_diStartStep,
    i_stReaction := iq_stStandardModuleItf.i_stReaction,
    iq_stExceptionList := iq_stExceptionList,
    iq_stLogDataList := iq_stLogDataList); // TPL.FB_LOGGER
END_ACTION

ACTION ModuleFaults:
(* System generated code, could be modified for your application *)
(* User Exception *)
fbExceptionHandler.SetException(	i_xExceptionActive	:= xModuleUserException1,
									iq_stException		:= stUserException1,
									iq_stExceptionList	:= iq_stExceptionList,
									q_etDiag			=> ,
									q_etDiagExt			=> ,
									q_sMsg				=> );

(* User Exception *)
fbExceptionHandler.SetException(	i_xExceptionActive	:= xModuleUserException2,
									iq_stException		:= stUserException2,
									iq_stExceptionList	:= iq_stExceptionList,
									q_etDiag			=> ,
									q_etDiagExt			=> ,
									q_sMsg				=> );

(* end of System generated code, could be modified for your application *)
END_ACTION

ACTION Output_Active:
(* System generated code, only to be changed by experienced programmers *)
IF iq_stStandardModuleItf.q_udiSubModuleInException <> 0 THEN
	iq_stStandardModuleItf.q_etDiag		:= GD.ET_Diag.Ok;
	iq_stStandardModuleItf.q_udiDiagExt	:= ET_DiagExt.SubModuleInException;
	iq_stStandardModuleItf.q_sDiagExt		:= FC_EtDiagExtToString(i_etDiagExt := ET_DiagExt.SubModuleInException);
	iq_stStandardModuleItf.q_sMsg			:= '';
ELSE
	IF etDiagModuleController = GD.ET_Diag.Ok THEN
		iq_stStandardModuleItf.q_etDiag	:= etDiagModuleController;
		iq_stStandardModuleItf.q_sMsg		:= sMsgModuleController;
		
		CASE etDiagExtModuleController OF
			TPL.ET_DiagExt.DeactivatingSubModules : 
				iq_stStandardModuleItf.q_udiDiagExt	:= ET_DiagExt.DeactivatingSubModules;
				iq_stStandardModuleItf.q_sDiagExt		:= FC_EtDiagExtToString(i_etDiagExt := ET_DiagExt.DeactivatingSubModules);
			TPL.ET_DiagExt.Disabled : 
				iq_stStandardModuleItf.q_udiDiagExt	:= ET_DiagExt.Disabled;
				iq_stStandardModuleItf.q_sDiagExt		:= FC_EtDiagExtToString(i_etDiagExt := ET_DiagExt.Disabled);
			TPL.ET_DiagExt.ExecuteStep : 
				iq_stStandardModuleItf.q_udiDiagExt	:= ET_DiagExt.ExecuteStep;
				iq_stStandardModuleItf.q_sDiagExt		:= FC_EtDiagExtToString(i_etDiagExt := ET_DiagExt.ExecuteStep);
			TPL.ET_DiagExt.Initializing : 
				iq_stStandardModuleItf.q_udiDiagExt	:= ET_DiagExt.Initializing;
				iq_stStandardModuleItf.q_sDiagExt		:= FC_EtDiagExtToString(i_etDiagExt := ET_DiagExt.Initializing);
			TPL.ET_DiagExt.WaitAtNegativeStep : 
				iq_stStandardModuleItf.q_udiDiagExt	:= ET_DiagExt.WaitAtNegativeStep;
				iq_stStandardModuleItf.q_sDiagExt		:= FC_EtDiagExtToString(i_etDiagExt := ET_DiagExt.WaitAtNegativeStep);
			TPL.ET_DiagExt.WaitCmdsDone : 
				iq_stStandardModuleItf.q_udiDiagExt	:= ET_DiagExt.WaitCmdsDone;
				iq_stStandardModuleItf.q_sDiagExt		:= FC_EtDiagExtToString(i_etDiagExt := ET_DiagExt.WaitCmdsDone);
			TPL.ET_DiagExt.WaitForCmd : 
				iq_stStandardModuleItf.q_udiDiagExt	:= ET_DiagExt.WaitForCmd;
				iq_stStandardModuleItf.q_sDiagExt		:= FC_EtDiagExtToString(i_etDiagExt := ET_DiagExt.WaitForCmd);
			ELSE
				iq_stStandardModuleItf.q_etDiag		:= GD. ET_Diag.UnexpectedProgramBehavior;
				iq_stStandardModuleItf.q_udiDiagExt	:= ET_DiagExt.UnknownStateModuleController;
				iq_stStandardModuleItf.q_sDiagExt		:= FC_EtDiagExtToString(i_etDiagExt := ET_DiagExt.UnknownStateModuleController);
		END_CASE
	ELSE
		iq_stStandardModuleItf.q_etDiag		:= GD.ET_Diag.DiagActive;
		iq_stStandardModuleItf.q_udiDiagExt	:= ET_DiagExt.ModuleControllerException;
		iq_stStandardModuleItf.q_sDiagExt	:= FC_EtDiagExtToString(i_etDiagExt := ET_DiagExt.ModuleControllerException);
		iq_stStandardModuleItf.q_sMsg		:= PDL.FC_MultiConcat(	i_sString1 := GD.FC_EtDiagToString(i_etDiag := etDiagModuleController), 
																	i_sString2 := ' - ',
																	i_sString3 := TPL.FC_EtDiagExtToString(i_etDiagExt := etDiagExtModuleController), 
																	i_sString4 := '');
	END_IF
END_IF

(* End of system generated code, only to be changed by experienced programmers *)
END_ACTION

METHOD RegisterLoggerPoint
VAR_INPUT
	i_ifParent	: APL.IF_LoggerPoint;
	i_sName		: STRING[80];
END_VAR
VAR_OUTPUT
	q_etDiag	: GD.ET_Diag := GD.ET_Diag.Ok;
	q_etDiagExt	: ET_DiagExt := ET_DiagExt.Ok;
END_VAR
fbLoggerPoint.RegisterLoggerPoint(	i_ifParent	:= i_ifParent,
									i_sName		:= i_sName,
									i_sType		:= 'Node Module',
									i_sSource	:= 'Program',
									q_etDiag	=> ,
									q_etDiagExt	=> );
END_METHOD

ACTION SubModules_Action:
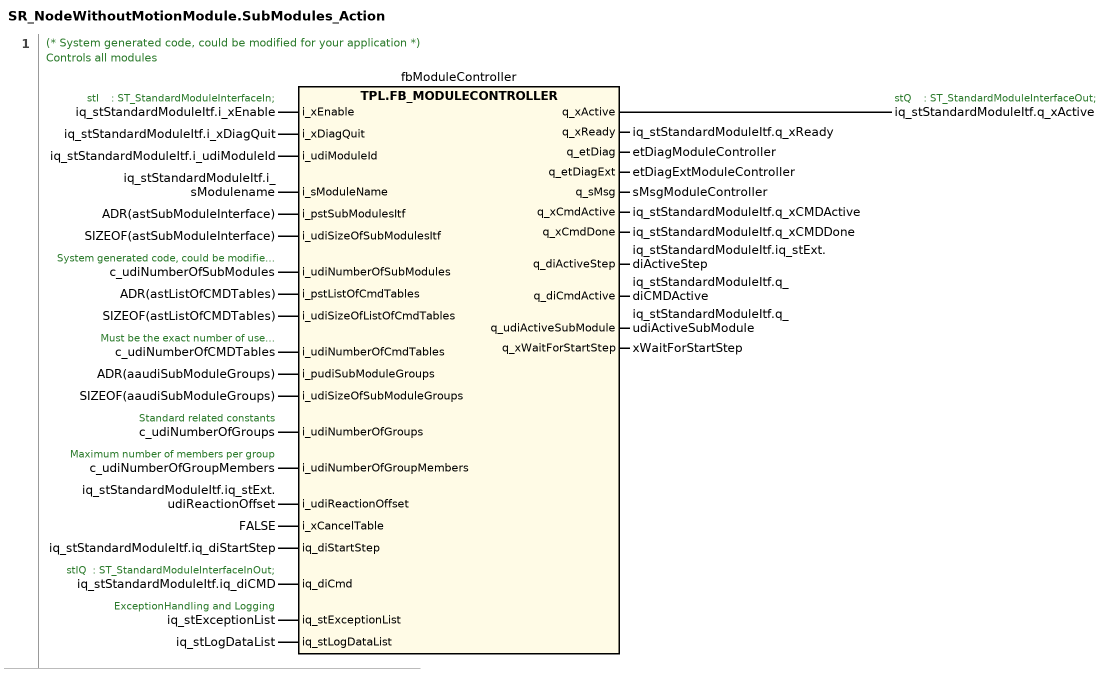
// NETWORK 1
// 					(* System generated code, could be modified for your application *)
// Controls all modules
//
//   fbModuleController: Modules related variables
//   iq_stStandardModuleItf.i_xEnable: stI : ST_StandardModuleInterfaceIn;
//   c_udiNumberOfSubModules: System generated code, could be modified for your application
//   c_udiNumberOfCMDTables: Must be the exact number of used CMDTables!
//   c_udiNumberOfGroups: Standard related constants
//   c_udiNumberOfGroupMembers: Maximum number of members per group
//   iq_stStandardModuleItf.iq_diCMD: stIQ : ST_StandardModuleInterfaceInOut;
//   iq_stExceptionList: ExceptionHandling and Logging
//   iq_stStandardModuleItf.q_xActive: stQ : ST_StandardModuleInterfaceOut;
fbModuleController(
    i_xEnable := iq_stStandardModuleItf.i_xEnable,
    i_xDiagQuit := iq_stStandardModuleItf.i_xDiagQuit,
    i_udiModuleId := iq_stStandardModuleItf.i_udiModuleId,
    i_sModuleName := iq_stStandardModuleItf.i_sModulename,
    i_pstSubModulesItf := ADR(astSubModuleInterface),
    i_udiSizeOfSubModulesItf := SIZEOF(astSubModuleInterface),
    i_udiNumberOfSubModules := c_udiNumberOfSubModules,
    i_pstListOfCmdTables := ADR(astListOfCMDTables),
    i_udiSizeOfListOfCmdTables := SIZEOF(astListOfCMDTables),
    i_udiNumberOfCmdTables := c_udiNumberOfCMDTables,
    i_pudiSubModuleGroups := ADR(aaudiSubModuleGroups),
    i_udiSizeOfSubModuleGroups := SIZEOF(aaudiSubModuleGroups),
    i_udiNumberOfGroups := c_udiNumberOfGroups,
    i_udiNumberOfGroupMembers := c_udiNumberOfGroupMembers,
    i_udiReactionOffset := iq_stStandardModuleItf.iq_stExt.udiReactionOffset,
    i_xCancelTable := FALSE,
    iq_diStartStep := iq_stStandardModuleItf.iq_diStartStep,
    iq_diCmd := iq_stStandardModuleItf.iq_diCMD,
    iq_stExceptionList := iq_stExceptionList,
    iq_stLogDataList := iq_stLogDataList,
    q_xReady => iq_stStandardModuleItf.q_xReady,
    q_etDiag => etDiagModuleController,
    q_etDiagExt => etDiagExtModuleController,
    q_sMsg => sMsgModuleController,
    q_xCmdActive => iq_stStandardModuleItf.q_xCMDActive,
    q_xCmdDone => iq_stStandardModuleItf.q_xCMDDone,
    q_diActiveStep => iq_stStandardModuleItf.iq_stExt.diActiveStep,
    q_diCmdActive => iq_stStandardModuleItf.q_diCMDActive,
    q_udiActiveSubModule => iq_stStandardModuleItf.q_udiActiveSubModule,
    q_xWaitForStartStep => xWaitForStartStep); // TPL.FB_MODULECONTROLLER
iq_stStandardModuleItf.q_xActive := fbModuleController.q_xActive;
END_ACTION

ACTION UpdateStructs:
(* System generated code, do not change without consulting 'Schneider Electric Automation GmbH' - otherwise you risk instability!!!*)
fbDetectOnlineChange(	i_xEnable	:= TRUE, 
						i_xDetect	:= TRUE, 
						q_xActive	=> xDetectOnlineChangeActive, 
						q_xReady	=> xDetectOnlineChangeReady, 
						q_etDiag	=> etDetectOnlineChangeDiag, 
						q_etDiagExt	=> etDetectOnlineChangeDiagExt, 
						q_sMsg		=> sDetectOnlineChangeMsg, 
						q_xChange	=> );
						
IF(NOT fbDetectOnlineChange.q_xChange) THEN
	RETURN;
END_IF

iq_stStandardModuleItf.iq_stExt.udiNumberOfSubModules 		:= c_udiNumberOfSubModules;
iq_stStandardModuleItf.iq_stExt.dwSubModulesItf		 		:= ADR(astSubModuleInterface);
iq_stStandardModuleItf.iq_stExt.pdwSubModulesAddItf		 	:= ADR(adwSubModuleAddInterfaces);
iq_stStandardModuleItf.iq_stExt.pstListofCMDTables			:= ADR(astListOfCMDTables);
iq_stStandardModuleItf.iq_stExt.udiNumberOfCmdTables		:= c_udiNumberOfCMDTables;
(* End of system generated code, do not change without consulting 'Schneider Electric Automation GmbH' - otherwise you risk instability!!!*)

(* System generated code, could be modified for your application *)
xUpdateStructsException := FALSE;

(*****************************************************************************************************************************************************)
(* Update CmdTable - Prepare *)

TPL.FC_UpdateCmdTableListElement(	i_pstListofCMDTables	:= ADR(astListofCMDTables),
									i_udiNumberOfCMDTables	:= c_udiNumberOfCMDTables,
									i_diCMD					:= ET_Cmd.Prepare,
									i_pstCMDTable			:= ADR(astPrepareTable),
									q_etDiag				=> etDiag,
									q_etDiagExt				=> etDiagExtTPL);
									
IF etDiag <> GD.ET_Diag.Ok AND NOT xUpdateStructsException THEN
	xUpdateStructsException := TRUE;
	
	stUpdateStructsException.sMsg := PDL.FC_MultiConcat(i_sString1 := 'Update CmdTable: Prepare - ', 
														i_sString2 := GD.FC_EtDiagToString(i_etDiag := etDiag), 
														i_sString3 := ' - ', 
														i_sString4 := TPL.FC_EtDiagExtToString(i_etDiagExt := etDiagExtTPL));
END_IF										

(*****************************************************************************************************************************************************)
(* Update CmdTable - Auto *)

TPL.FC_UpdateCmdTableListElement(	i_pstListofCMDTables	:= ADR(astListofCMDTables),
									i_udiNumberOfCMDTables	:= c_udiNumberOfCMDTables,
									i_diCMD					:= ET_Cmd.Auto,
									i_pstCMDTable			:= ADR(astAutoTable),
									q_etDiag				=> etDiag,
									q_etDiagExt				=> etDiagExtTPL);
									
IF etDiag <> GD.ET_Diag.Ok AND NOT xUpdateStructsException THEN
	xUpdateStructsException := TRUE;
	
	stUpdateStructsException.sMsg := PDL.FC_MultiConcat(i_sString1 := 'Update CmdTable: Auto - ', 
														i_sString2 := GD.FC_EtDiagToString(i_etDiag := etDiag), 
														i_sString3 := ' - ', 
														i_sString4 := TPL.FC_EtDiagExtToString(i_etDiagExt := etDiagExtTPL));
END_IF		

(*****************************************************************************************************************************************************)
(* Update CmdTable - Manual *)

TPL.FC_UpdateCmdTableListElement(	i_pstListofCMDTables	:= ADR(astListofCMDTables),
									i_udiNumberOfCMDTables	:= c_udiNumberOfCMDTables,
									i_diCMD					:= ET_Cmd.Manual,
									i_pstCMDTable			:= ADR(astManualTable),
									q_etDiag				=> etDiag,
									q_etDiagExt				=> etDiagExtTPL);
									
IF etDiag <> GD.ET_Diag.Ok AND NOT xUpdateStructsException THEN
	xUpdateStructsException := TRUE;
	
	stUpdateStructsException.sMsg := PDL.FC_MultiConcat(i_sString1 := 'Update CmdTable: Manual - ', 
														i_sString2 := GD.FC_EtDiagToString(i_etDiag := etDiag), 
														i_sString3 := ' - ', 
														i_sString4 := TPL.FC_EtDiagExtToString(i_etDiagExt := etDiagExtTPL));
END_IF		

(*****************************************************************************************************************************************************)
(* Update CmdTable - Stop *)

TPL.FC_UpdateCmdTableListElement(	i_pstListofCMDTables	:= ADR(astListofCMDTables),
									i_udiNumberOfCMDTables	:= c_udiNumberOfCMDTables,
									i_diCMD					:= ET_Cmd.Stop,
									i_pstCMDTable			:= ADR(astStopTable),
									q_etDiag				=> etDiag,
									q_etDiagExt				=> etDiagExtTPL);
									
IF etDiag <> GD.ET_Diag.Ok AND NOT xUpdateStructsException THEN
	xUpdateStructsException := TRUE;
	
	stUpdateStructsException.sMsg := PDL.FC_MultiConcat(i_sString1 := 'Update CmdTable: Stop - ', 
														i_sString2 := GD.FC_EtDiagToString(i_etDiag := etDiag), 
														i_sString3 := ' - ', 
														i_sString4 := TPL.FC_EtDiagExtToString(i_etDiagExt := etDiagExtTPL));
END_IF		

(*****************************************************************************************************************************************************)
(* Update CmdTable - Start *)

TPL.FC_UpdateCmdTableListElement(	i_pstListofCMDTables	:= ADR(astListofCMDTables),
									i_udiNumberOfCMDTables	:= c_udiNumberOfCMDTables,
									i_diCMD					:= ET_Cmd.Start,
									i_pstCMDTable			:= ADR(astStartTable),
									q_etDiag				=> etDiag,
									q_etDiagExt				=> etDiagExtTPL);
									
IF etDiag <> GD.ET_Diag.Ok AND NOT xUpdateStructsException THEN
	xUpdateStructsException := TRUE;
	
	stUpdateStructsException.sMsg := PDL.FC_MultiConcat(i_sString1 := 'Update CmdTable: Start - ', 
														i_sString2 := GD.FC_EtDiagToString(i_etDiag := etDiag), 
														i_sString3 := ' - ', 
														i_sString4 := TPL.FC_EtDiagExtToString(i_etDiagExt := etDiagExtTPL));
END_IF		

(*****************************************************************************************************************************************************)
(* Update CmdTable - Abort *)

TPL.FC_UpdateCmdTableListElement(	i_pstListofCMDTables	:= ADR(astListofCMDTables),
									i_udiNumberOfCMDTables	:= c_udiNumberOfCMDTables,
									i_diCMD					:= ET_Cmd.Abort,
									i_pstCMDTable			:= ADR(astAbortTable),
									q_etDiag				=> etDiag,
									q_etDiagExt				=> etDiagExtTPL);
									
IF etDiag <> GD.ET_Diag.Ok AND NOT xUpdateStructsException THEN
	xUpdateStructsException := TRUE;
	
	stUpdateStructsException.sMsg := PDL.FC_MultiConcat(i_sString1 := 'Update CmdTable: Abort - ', 
														i_sString2 := GD.FC_EtDiagToString(i_etDiag := etDiag), 
														i_sString3 := ' - ', 
														i_sString4 := TPL.FC_EtDiagExtToString(i_etDiagExt := etDiagExtTPL));
END_IF		

(*****************************************************************************************************************************************************)
(* Update CmdTable - Hold *)

TPL.FC_UpdateCmdTableListElement(	i_pstListofCMDTables	:= ADR(astListofCMDTables),
									i_udiNumberOfCMDTables	:= c_udiNumberOfCMDTables,
									i_diCMD					:= ET_Cmd.Hold,
									i_pstCMDTable			:= ADR(astHoldTable),
									q_etDiag				=> etDiag,
									q_etDiagExt				=> etDiagExtTPL);
									
IF etDiag <> GD.ET_Diag.Ok AND NOT xUpdateStructsException THEN
	xUpdateStructsException := TRUE;
	
	stUpdateStructsException.sMsg := PDL.FC_MultiConcat(i_sString1 := 'Update CmdTable: Hold - ', 
														i_sString2 := GD.FC_EtDiagToString(i_etDiag := etDiag), 
														i_sString3 := ' - ', 
														i_sString4 := TPL.FC_EtDiagExtToString(i_etDiagExt := etDiagExtTPL));
END_IF		

(*****************************************************************************************************************************************************)
(* Update CmdTable - BrakeRelease *)

TPL.FC_UpdateCmdTableListElement(	i_pstListofCMDTables	:= ADR(astListofCMDTables),
									i_udiNumberOfCMDTables	:= c_udiNumberOfCMDTables,
									i_diCMD					:= ET_Cmd.BrakeRelease,
									i_pstCMDTable			:= ADR(astBrakeReleaseTable),
									q_etDiag				=> etDiag,
									q_etDiagExt				=> etDiagExtTPL);
									
IF etDiag <> GD.ET_Diag.Ok AND NOT xUpdateStructsException THEN
	xUpdateStructsException := TRUE;
	
	stUpdateStructsException.sMsg := PDL.FC_MultiConcat(i_sString1 := 'Update CmdTable: BrakeRelease - ', 
														i_sString2 := GD.FC_EtDiagToString(i_etDiag := etDiag), 
														i_sString3 := ' - ', 
														i_sString4 := TPL.FC_EtDiagExtToString(i_etDiagExt := etDiagExtTPL));
END_IF		

(*****************************************************************************************************************************************************)
(* Set exception if any exception occurred *)

fbExceptionHandler.SetException(i_xExceptionActive	:= xUpdateStructsException, 
								iq_stException		:= stUpdateStructsException, 
								iq_stExceptionList	:= iq_stExceptionList);
					
xInitSuccessful := xInitSuccessful AND NOT xUpdateStructsException;

etDiag := GD.ET_Diag.Ok;
(* End of system generated code, could be modified for your application *)
END_ACTION

END_PROGRAM

// LMC_PacDrive/Application/FC_ObjectTypeIsMotionAxis
(* Checks whether the given diObjectType is an object representing a Motion Axis (drive beneath SercosIII bus) *)
FUNCTION FC_ObjectTypeIsMotionAxis : BOOL

VAR_INPUT
	i_udiObjectType: UDINT; (* Type (UDINT) of object to be checked to be a motion axis *)  
END_VAR

(* Currently, this implemetation is hacky. We compare the ObjectType to a static list of ObjectTypes known as Motion Drives.
   What we acutlly want is to get the IEC object by LogicalAddress and check whether it fits the interface IF_Drive. But sadly, 
   such a function doesn't exist yet *)

IF	i_udiObjectType = SystemInterface.LXM62DxS_TYPE.udiType OR
	i_udiObjectType = SystemInterface.ILM62_TYPE.udiType OR
	i_udiObjectType = SystemInterface.LXM52_TYPE.udiType OR
	i_udiObjectType = SystemInterface.SERCDRV_TYPE.udiType OR
	i_udiObjectType = SystemInterface.LXM52Linear_TYPE.udiType OR
	i_udiObjectType = SystemInterface.LXM62DxSLinear_TYPE.udiType
THEN
   FC_ObjectTypeIsMotionAxis := TRUE;
ELSE
   FC_ObjectTypeIsMotionAxis := FALSE;
END_IF

RETURN;

END_FUNCTION

